Yaskawa INFORM job: A_ROOF_SIDE_0617_2_PAINT_50.JBI

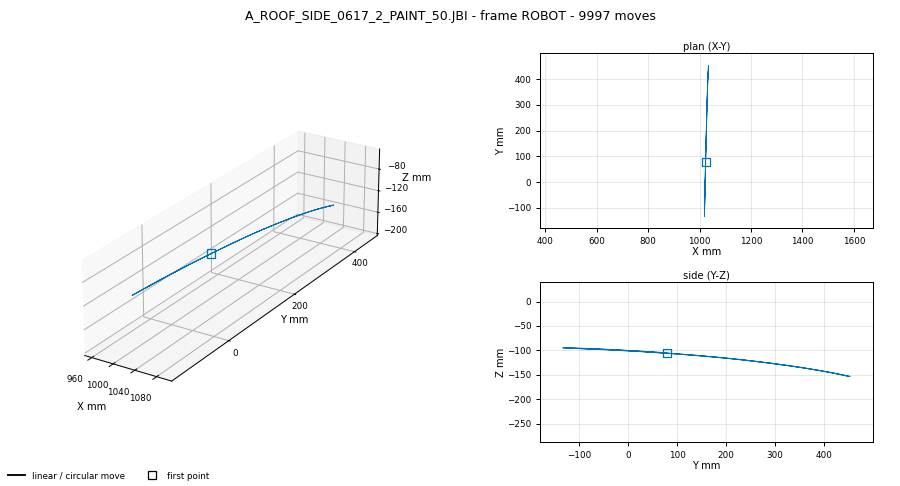
[picture p0: tool path of A_ROOF_SIDE_0617_2_PAINT_50.JBI in frame ROBOT, 9997 of 9997 moves have a stored position in this frame; points joined in program order, loops and branches not executed]
/JOB
//NAME A_ROOF_SIDE_0617_2_PAINT50
//POS
///NPOS 9997,0,0,0,0,0
///TOOL 1
///USER 0
///POSTYPE ROBOT
///RECTAN
///RCONF 1,0,0,0,0,0,0,0,0,0,0,0,0,0,0,0,0,0,0,0,0,0,0,0
C00000=1024.133,78.884,-104.654,167.721,48.501,158.989
C00001=1024.128,78.635,-104.636,167.719,48.505,158.990
C00002=1024.122,78.385,-104.618,167.716,48.509,158.990
C00003=1024.116,78.136,-104.601,167.715,48.513,158.991
C00004=1024.111,77.886,-104.582,167.712,48.517,158.991
C00005=1024.105,77.637,-104.565,167.709,48.522,158.992
C00006=1024.099,77.389,-104.548,167.707,48.526,158.992
C00007=1024.093,77.139,-104.530,167.704,48.530,158.992
C00008=1024.087,76.890,-104.512,167.702,48.535,158.993
C00009=1024.081,76.640,-104.494,167.699,48.539,158.993
C00010=1024.076,76.391,-104.477,167.697,48.543,158.994
C00011=1024.069,76.141,-104.459,167.694,48.547,158.994
C00012=1024.063,75.858,-104.439,167.690,48.552,158.995
C00013=1024.056,75.573,-104.419,167.687,48.558,158.995
C00014=1024.049,75.289,-104.400,167.685,48.562,158.996
C00015=1024.042,75.005,-104.379,167.681,48.567,158.996
C00016=1024.037,74.756,-104.362,167.679,48.572,158.997
C00017=1024.030,74.506,-104.345,167.676,48.576,158.997
C00018=1024.025,74.257,-104.327,167.674,48.580,158.998
C00019=1024.018,74.008,-104.309,167.671,48.585,158.998
C00020=1024.013,73.759,-104.291,167.668,48.589,158.999
C00021=1024.007,73.509,-104.275,167.666,48.593,158.999
C00022=1024.001,73.260,-104.257,167.663,48.597,158.999
C00023=1023.995,73.010,-104.240,167.661,48.602,159.000
C00024=1023.989,72.761,-104.222,167.658,48.606,159.000
C00025=1023.983,72.512,-104.205,167.655,48.610,159.001
C00026=1023.977,72.263,-104.187,167.653,48.614,159.001
C00027=1023.972,72.013,-104.170,167.650,48.619,159.002
C00028=1023.965,71.764,-104.153,167.648,48.623,159.002
C00029=1023.960,71.515,-104.135,167.645,48.627,159.003
C00030=1023.954,71.265,-104.118,167.643,48.632,159.003
C00031=1023.948,71.016,-104.101,167.640,48.636,159.003
C00032=1023.942,70.767,-104.084,167.637,48.640,159.004
C00033=1023.936,70.517,-104.066,167.635,48.644,159.004
C00034=1023.931,70.268,-104.048,167.632,48.649,159.005
C00035=1023.924,70.019,-104.031,167.629,48.653,159.005
C00036=1023.919,69.769,-104.014,167.627,48.657,159.006
C00037=1023.913,69.520,-103.996,167.624,48.661,159.006
C00038=1023.907,69.271,-103.979,167.622,48.666,159.007
C00039=1023.901,69.021,-103.962,167.619,48.670,159.007
C00040=1023.895,68.772,-103.945,167.618,48.674,159.008
C00041=1023.889,68.523,-103.928,167.615,48.678,159.008
C00042=1023.883,68.273,-103.911,167.612,48.682,159.008
C00043=1023.877,68.024,-103.894,167.609,48.687,159.009
C00044=1023.872,67.775,-103.876,167.606,48.691,159.009
C00045=1023.866,67.525,-103.860,167.604,48.696,159.010
C00046=1023.860,67.276,-103.842,167.601,48.700,159.010
C00047=1023.854,67.027,-103.824,167.599,48.704,159.011
C00048=1023.848,66.777,-103.808,167.596,48.709,159.011
C00049=1023.842,66.528,-103.790,167.593,48.713,159.011
C00050=1023.836,66.278,-103.774,167.591,48.717,159.012
C00051=1023.830,66.029,-103.756,167.588,48.721,159.012
C00052=1023.824,65.780,-103.739,167.586,48.726,159.013
C00053=1023.818,65.530,-103.722,167.583,48.730,159.013
C00054=1023.812,65.281,-103.705,167.581,48.734,159.014
C00055=1023.807,65.032,-103.688,167.578,48.738,159.014
C00056=1023.800,64.782,-103.671,167.575,48.743,159.015
C00057=1023.795,64.533,-103.654,167.573,48.748,159.015
C00058=1023.789,64.284,-103.637,167.570,48.752,159.015
C00059=1023.783,64.034,-103.620,167.568,48.756,159.016
C00060=1023.777,63.785,-103.603,167.565,48.760,159.016
C00061=1023.771,63.535,-103.586,167.563,48.765,159.017
C00062=1023.765,63.286,-103.569,167.560,48.769,159.017
C00063=1023.759,63.036,-103.552,167.557,48.773,159.018
C00064=1023.753,62.787,-103.536,167.555,48.778,159.018
C00065=1023.747,62.538,-103.519,167.552,48.782,159.019
C00066=1023.741,62.289,-103.502,167.550,48.786,159.019
C00067=1023.734,62.039,-103.485,167.547,48.791,159.020
C00068=1023.728,61.790,-103.469,167.545,48.796,159.020
C00069=1023.723,61.540,-103.452,167.542,48.799,159.020
C00070=1023.717,61.291,-103.435,167.540,48.804,159.021
C00071=1023.710,61.041,-103.418,167.537,48.809,159.022
C00072=1023.704,60.792,-103.402,167.535,48.813,159.022
C00073=1023.698,60.543,-103.385,167.532,48.817,159.022
C00074=1023.693,60.294,-103.368,167.530,48.822,159.023
C00075=1023.687,60.044,-103.352,167.527,48.826,159.023
C00076=1023.680,59.759,-103.333,167.524,48.831,159.024
C00077=1023.673,59.476,-103.314,167.520,48.836,159.024
C00078=1023.666,59.191,-103.295,167.518,48.841,159.025
C00079=1023.659,58.907,-103.276,167.515,48.846,159.025
C00080=1023.653,58.658,-103.259,167.512,48.850,159.026
C00081=1023.647,58.408,-103.242,167.510,48.855,159.026
C00082=1023.641,58.159,-103.226,167.507,48.860,159.027
C00083=1023.635,57.909,-103.210,167.505,48.864,159.027
C00084=1023.629,57.660,-103.192,167.502,48.868,159.028
C00085=1023.623,57.411,-103.176,167.499,48.872,159.028
C00086=1023.617,57.162,-103.160,167.497,48.877,159.029
C00087=1023.611,56.912,-103.143,167.495,48.881,159.029
C00088=1023.604,56.663,-103.126,167.492,48.885,159.029
C00089=1023.598,56.413,-103.110,167.489,48.890,159.030
C00090=1023.593,56.164,-103.093,167.486,48.895,159.030
C00091=1023.587,55.914,-103.077,167.483,48.899,159.031
C00092=1023.581,55.665,-103.061,167.481,48.903,159.031
C00093=1023.575,55.416,-103.044,167.478,48.907,159.032
C00094=1023.569,55.166,-103.027,167.476,48.912,159.032
C00095=1023.563,54.917,-103.011,167.473,48.917,159.033
C00096=1023.557,54.667,-102.994,167.470,48.921,159.033
C00097=1023.551,54.418,-102.978,167.468,48.925,159.033
C00098=1023.546,54.169,-102.961,167.465,48.929,159.034
C00099=1023.539,53.920,-102.944,167.463,48.934,159.034
C00100=1023.533,53.671,-102.928,167.460,48.938,159.035
C00101=1023.527,53.421,-102.912,167.458,48.942,159.035
C00102=1023.522,53.172,-102.895,167.455,48.946,159.036
C00103=1023.516,52.921,-102.878,167.453,48.951,159.036
C00104=1023.510,52.672,-102.862,167.450,48.955,159.037
C00105=1023.504,52.423,-102.846,167.447,48.959,159.037
C00106=1023.498,52.173,-102.830,167.445,48.964,159.037
C00107=1023.492,51.924,-102.813,167.442,48.968,159.038
C00108=1023.486,51.675,-102.796,167.440,48.973,159.038
C00109=1023.480,51.426,-102.780,167.437,48.977,159.039
C00110=1023.474,51.176,-102.763,167.435,48.981,159.039
C00111=1023.468,50.927,-102.747,167.432,48.985,159.040
C00112=1023.462,50.678,-102.731,167.430,48.990,159.040
C00113=1023.457,50.428,-102.715,167.427,48.994,159.040
C00114=1023.451,50.179,-102.698,167.424,48.998,159.041
C00115=1023.445,49.929,-102.681,167.422,49.002,159.041
C00116=1023.439,49.680,-102.665,167.419,49.007,159.042
C00117=1023.433,49.431,-102.649,167.416,49.011,159.042
C00118=1023.427,49.181,-102.633,167.414,49.016,159.043
C00119=1023.422,48.932,-102.616,167.411,49.019,159.043
C00120=1023.416,48.683,-102.600,167.409,49.024,159.043
C00121=1023.410,48.433,-102.584,167.406,49.028,159.044
C00122=1023.404,48.184,-102.567,167.403,49.032,159.044
C00123=1023.398,47.934,-102.551,167.401,49.037,159.045
C00124=1023.393,47.685,-102.535,167.398,49.041,159.045
C00125=1023.387,47.435,-102.518,167.396,49.045,159.046
C00126=1023.381,47.186,-102.502,167.393,49.049,159.046
C00127=1023.375,46.937,-102.486,167.391,49.054,159.046
C00128=1023.369,46.687,-102.470,167.388,49.058,159.047
C00129=1023.364,46.438,-102.453,167.386,49.062,159.047
C00130=1023.358,46.188,-102.436,167.383,49.066,159.048
C00131=1023.352,45.939,-102.420,167.380,49.070,159.048
C00132=1023.346,45.690,-102.404,167.378,49.075,159.048
C00133=1023.340,45.440,-102.388,167.375,49.079,159.049
C00134=1023.334,45.191,-102.371,167.373,49.084,159.049
C00135=1023.328,44.942,-102.355,167.370,49.087,159.050
C00136=1023.322,44.692,-102.339,167.368,49.091,159.050
C00137=1023.317,44.443,-102.322,167.366,49.096,159.051
C00138=1023.311,44.193,-102.306,167.363,49.100,159.051
C00139=1023.305,43.943,-102.290,167.360,49.104,159.051
C00140=1023.299,43.659,-102.272,167.357,49.109,159.052
C00141=1023.292,43.375,-102.253,167.354,49.113,159.052
C00142=1023.285,43.089,-102.235,167.351,49.118,159.053
C00143=1023.279,42.805,-102.216,167.349,49.123,159.053
C00144=1023.273,42.556,-102.200,167.346,49.128,159.054
C00145=1023.267,42.307,-102.184,167.344,49.132,159.054
C00146=1023.261,42.057,-102.168,167.341,49.136,159.054
C00147=1023.254,41.808,-102.152,167.337,49.140,159.055
C00148=1023.249,41.558,-102.136,167.335,49.145,159.055
C00149=1023.243,41.309,-102.120,167.332,49.149,159.056
C00150=1023.237,41.059,-102.104,167.330,49.154,159.056
C00151=1023.232,40.810,-102.088,167.327,49.158,159.056
C00152=1023.226,40.561,-102.072,167.325,49.162,159.057
C00153=1023.220,40.311,-102.057,167.322,49.166,159.057
C00154=1023.213,40.062,-102.041,167.320,49.171,159.058
C00155=1023.207,39.813,-102.025,167.317,49.175,159.058
C00156=1023.202,39.563,-102.009,167.315,49.180,159.059
C00157=1023.196,39.313,-101.993,167.312,49.183,159.059
C00158=1023.190,39.064,-101.977,167.309,49.188,159.059
C00159=1023.184,38.814,-101.961,167.307,49.192,159.060
C00160=1023.178,38.566,-101.946,167.304,49.197,159.060
C00161=1023.172,38.316,-101.930,167.302,49.201,159.061
C00162=1023.166,38.066,-101.914,167.299,49.205,159.061
C00163=1023.161,37.817,-101.898,167.296,49.209,159.062
C00164=1023.155,37.568,-101.881,167.294,49.213,159.062
C00165=1023.149,37.318,-101.866,167.291,49.218,159.062
C00166=1023.142,37.069,-101.850,167.289,49.222,159.063
C00167=1023.137,36.819,-101.835,167.286,49.227,159.063
C00168=1023.131,36.570,-101.819,167.283,49.231,159.064
C00169=1023.126,36.320,-101.803,167.281,49.235,159.064
C00170=1023.119,36.071,-101.788,167.278,49.239,159.064
C00171=1023.113,35.821,-101.772,167.276,49.244,159.065
C00172=1023.107,35.572,-101.756,167.274,49.249,159.065
C00173=1023.101,35.322,-101.741,167.271,49.253,159.066
C00174=1023.096,35.073,-101.725,167.268,49.257,159.066
C00175=1023.089,34.824,-101.710,167.265,49.261,159.067
C00176=1023.083,34.574,-101.694,167.262,49.266,159.067
C00177=1023.077,34.325,-101.679,167.260,49.270,159.067
C00178=1023.071,34.075,-101.663,167.257,49.275,159.068
C00179=1023.066,33.826,-101.647,167.255,49.279,159.068
C00180=1023.059,33.576,-101.632,167.252,49.283,159.069
C00181=1023.054,33.327,-101.616,167.249,49.287,159.069
C00182=1023.047,33.077,-101.601,167.247,49.292,159.070
C00183=1023.041,32.828,-101.585,167.244,49.296,159.070
C00184=1023.035,32.579,-101.570,167.242,49.301,159.070
C00185=1023.029,32.330,-101.554,167.239,49.305,159.071
C00186=1023.024,32.080,-101.539,167.237,49.309,159.071
C00187=1023.017,31.830,-101.524,167.234,49.313,159.072
C00188=1023.011,31.581,-101.507,167.232,49.318,159.072
C00189=1023.006,31.332,-101.493,167.229,49.322,159.072
C00190=1023.000,31.082,-101.477,167.227,49.327,159.073
C00191=1022.994,30.832,-101.461,167.224,49.331,159.073
C00192=1022.988,30.583,-101.446,167.221,49.336,159.074
C00193=1022.983,30.334,-101.431,167.218,49.340,159.074
C00194=1022.976,30.085,-101.415,167.215,49.344,159.075
C00195=1022.970,29.835,-101.400,167.213,49.348,159.075
C00196=1022.965,29.585,-101.384,167.210,49.352,159.075
C00197=1022.959,29.336,-101.369,167.208,49.357,159.076
C00198=1022.953,29.086,-101.353,167.205,49.361,159.076
C00199=1022.947,28.837,-101.338,167.203,49.366,159.077
C00200=1022.941,28.587,-101.322,167.200,49.370,159.077
C00201=1022.935,28.338,-101.308,167.197,49.374,159.077
C00202=1022.929,28.088,-101.292,167.195,49.378,159.078
C00203=1022.923,27.839,-101.276,167.192,49.382,159.078
C00204=1022.916,27.554,-101.258,167.189,49.387,159.078
C00205=1022.910,27.269,-101.242,167.187,49.393,159.079
C00206=1022.903,26.985,-101.225,167.183,49.398,159.080
C00207=1022.896,26.700,-101.207,167.180,49.403,159.080
C00208=1022.890,26.452,-101.191,167.177,49.407,159.080
C00209=1022.884,26.202,-101.176,167.175,49.411,159.081
C00210=1022.878,25.952,-101.161,167.172,49.415,159.081
C00211=1022.873,25.703,-101.146,167.170,49.420,159.082
C00212=1022.866,25.453,-101.131,167.167,49.424,159.082
C00213=1022.861,25.204,-101.116,167.165,49.429,159.083
C00214=1022.854,24.954,-101.101,167.162,49.433,159.083
C00215=1022.848,24.705,-101.086,167.159,49.437,159.083
C00216=1022.843,24.456,-101.070,167.157,49.441,159.084
C00217=1022.836,24.206,-101.055,167.153,49.446,159.084
C00218=1022.830,23.957,-101.041,167.151,49.450,159.084
C00219=1022.825,23.707,-101.025,167.148,49.455,159.085
C00220=1022.818,23.457,-101.010,167.146,49.459,159.085
C00221=1022.813,23.208,-100.995,167.143,49.464,159.086
C00222=1022.807,22.958,-100.980,167.140,49.468,159.086
C00223=1022.801,22.709,-100.965,167.138,49.472,159.087
C00224=1022.795,22.460,-100.950,167.135,49.476,159.087
C00225=1022.789,22.210,-100.935,167.133,49.481,159.087
C00226=1022.783,21.961,-100.920,167.130,49.485,159.088
C00227=1022.777,21.711,-100.905,167.128,49.490,159.088
C00228=1022.771,21.461,-100.890,167.124,49.494,159.089
C00229=1022.765,21.212,-100.875,167.122,49.498,159.089
C00230=1022.759,20.963,-100.860,167.119,49.503,159.089
C00231=1022.753,20.714,-100.846,167.116,49.507,159.090
C00232=1022.748,20.464,-100.830,167.114,49.511,159.090
C00233=1022.741,20.214,-100.815,167.111,49.515,159.091
C00234=1022.736,19.965,-100.801,167.109,49.519,159.091
C00235=1022.730,19.715,-100.785,167.106,49.524,159.091
C00236=1022.724,19.466,-100.770,167.104,49.528,159.092
C00237=1022.718,19.216,-100.756,167.101,49.533,159.092
C00238=1022.712,18.967,-100.740,167.099,49.537,159.093
C00239=1022.706,18.718,-100.725,167.096,49.541,159.093
C00240=1022.700,18.468,-100.710,167.092,49.546,159.093
C00241=1022.694,18.219,-100.696,167.090,49.550,159.094
C00242=1022.688,17.969,-100.681,167.087,49.554,159.094
C00243=1022.682,17.720,-100.667,167.085,49.559,159.095
C00244=1022.677,17.470,-100.652,167.082,49.563,159.095
C00245=1022.670,17.220,-100.637,167.080,49.567,159.095
C00246=1022.664,16.971,-100.622,167.077,49.572,159.096
C00247=1022.658,16.721,-100.607,167.075,49.576,159.096
C00248=1022.652,16.473,-100.592,167.072,49.581,159.097
C00249=1022.647,16.222,-100.578,167.069,49.585,159.097
C00250=1022.641,15.973,-100.563,167.066,49.590,159.097
C00251=1022.635,15.723,-100.548,167.063,49.594,159.098
C00252=1022.629,15.474,-100.534,167.061,49.598,159.098
C00253=1022.623,15.225,-100.519,167.058,49.602,159.098
C00254=1022.617,14.975,-100.505,167.056,49.606,159.099
C00255=1022.611,14.725,-100.489,167.053,49.611,159.099
C00256=1022.606,14.476,-100.475,167.051,49.615,159.100
C00257=1022.599,14.227,-100.460,167.048,49.619,159.100
C00258=1022.594,13.978,-100.445,167.046,49.624,159.100
C00259=1022.587,13.727,-100.431,167.042,49.628,159.101
C00260=1022.582,13.478,-100.416,167.040,49.633,159.101
C00261=1022.575,13.229,-100.401,167.037,49.637,159.102
C00262=1022.570,12.979,-100.387,167.034,49.642,159.102
C00263=1022.563,12.729,-100.373,167.032,49.646,159.102
C00264=1022.558,12.481,-100.358,167.029,49.650,159.103
C00265=1022.552,12.230,-100.344,167.026,49.655,159.103
C00266=1022.546,11.981,-100.329,167.023,49.659,159.104
C00267=1022.540,11.731,-100.315,167.021,49.663,159.104
C00268=1022.533,11.448,-100.299,167.017,49.668,159.104
C00269=1022.526,11.165,-100.282,167.015,49.674,159.105
C00270=1022.519,10.882,-100.266,167.012,49.679,159.105
C00271=1022.512,10.599,-100.250,167.009,49.684,159.106
C00272=1022.506,10.349,-100.235,167.006,49.688,159.106
C00273=1022.500,10.100,-100.221,167.004,49.693,159.107
C00274=1022.494,9.850,-100.207,167.001,49.697,159.107
C00275=1022.488,9.601,-100.192,166.997,49.702,159.107
C00276=1022.481,9.351,-100.178,166.995,49.706,159.108
C00277=1022.476,9.102,-100.164,166.992,49.710,159.108
C00278=1022.470,8.853,-100.149,166.990,49.714,159.109
C00279=1022.464,8.603,-100.135,166.987,49.719,159.109
C00280=1022.458,8.354,-100.120,166.985,49.723,159.109
C00281=1022.452,8.103,-100.106,166.981,49.728,159.110
C00282=1022.446,7.854,-100.091,166.979,49.732,159.110
C00283=1022.440,7.604,-100.078,166.976,49.737,159.111
C00284=1022.434,7.355,-100.063,166.974,49.741,159.111
C00285=1022.428,7.106,-100.049,166.971,49.745,159.111
C00286=1022.422,6.856,-100.035,166.969,49.750,159.112
C00287=1022.417,6.607,-100.021,166.966,49.754,159.112
C00288=1022.410,6.356,-100.006,166.963,49.759,159.112
C00289=1022.405,6.107,-99.992,166.960,49.763,159.113
C00290=1022.398,5.858,-99.979,166.957,49.767,159.113
C00291=1022.392,5.608,-99.964,166.955,49.771,159.114
C00292=1022.387,5.359,-99.950,166.952,49.775,159.114
C00293=1022.381,5.110,-99.935,166.950,49.780,159.114
C00294=1022.375,4.860,-99.921,166.946,49.785,159.115
C00295=1022.369,4.610,-99.907,166.943,49.789,159.115
C00296=1022.364,4.361,-99.892,166.941,49.793,159.115
C00297=1022.357,4.111,-99.879,166.938,49.797,159.116
C00298=1022.351,3.862,-99.864,166.936,49.802,159.116
C00299=1022.345,3.613,-99.850,166.933,49.806,159.117
C00300=1022.339,3.362,-99.836,166.931,49.810,159.117
C00301=1022.334,3.113,-99.822,166.927,49.815,159.117
C00302=1022.328,2.864,-99.808,166.925,49.819,159.118
C00303=1022.322,2.614,-99.793,166.922,49.823,159.118
C00304=1022.316,2.365,-99.779,166.920,49.828,159.118
C00305=1022.310,2.115,-99.766,166.917,49.832,159.119
C00306=1022.304,1.865,-99.751,166.914,49.836,159.119
C00307=1022.298,1.616,-99.737,166.912,49.841,159.120
C00308=1022.293,1.367,-99.723,166.909,49.845,159.120
C00309=1022.287,1.117,-99.709,166.905,49.849,159.120
C00310=1022.281,0.867,-99.694,166.903,49.854,159.121
C00311=1022.275,0.618,-99.681,166.900,49.858,159.121
C00312=1022.269,0.368,-99.667,166.898,49.862,159.121
C00313=1022.263,0.118,-99.653,166.895,49.866,159.122
C00314=1022.257,-0.131,-99.638,166.893,49.871,159.122
C00315=1022.252,-0.380,-99.624,166.890,49.875,159.122
C00316=1022.246,-0.630,-99.610,166.886,49.879,159.123
C00317=1022.240,-0.880,-99.596,166.884,49.884,159.123
C00318=1022.234,-1.129,-99.582,166.881,49.888,159.123
C00319=1022.228,-1.378,-99.568,166.879,49.892,159.124
C00320=1022.223,-1.628,-99.555,166.876,49.896,159.124
C00321=1022.217,-1.878,-99.541,166.874,49.901,159.125
C00322=1022.211,-2.127,-99.526,166.871,49.905,159.125
C00323=1022.205,-2.377,-99.512,166.868,49.909,159.125
C00324=1022.199,-2.626,-99.499,166.866,49.913,159.125
C00325=1022.194,-2.876,-99.485,166.862,49.917,159.126
C00326=1022.188,-3.125,-99.471,166.860,49.922,159.126
C00327=1022.182,-3.375,-99.456,166.857,49.926,159.127
C00328=1022.176,-3.624,-99.442,166.854,49.930,159.127
C00329=1022.171,-3.874,-99.428,166.851,49.934,159.127
C00330=1022.165,-4.123,-99.415,166.849,49.939,159.128
C00331=1022.159,-4.374,-99.401,166.846,49.943,159.128
C00332=1022.152,-4.654,-99.385,166.843,49.948,159.128
C00333=1022.146,-4.936,-99.370,166.840,49.953,159.129
C00334=1022.139,-5.217,-99.355,166.836,49.958,159.129
C00335=1022.132,-5.499,-99.340,166.834,49.963,159.130
C00336=1022.126,-5.748,-99.326,166.830,49.967,159.130
C00337=1022.120,-5.997,-99.312,166.828,49.972,159.130
C00338=1022.114,-6.247,-99.299,166.825,49.976,159.131
C00339=1022.108,-6.497,-99.285,166.823,49.981,159.131
C00340=1022.102,-6.746,-99.272,166.819,49.985,159.131
C00341=1022.096,-6.996,-99.258,166.817,49.989,159.132
C00342=1022.090,-7.245,-99.244,166.814,49.994,159.132
C00343=1022.085,-7.495,-99.231,166.812,49.998,159.132
C00344=1022.078,-7.745,-99.217,166.809,50.003,159.133
C00345=1022.073,-7.994,-99.203,166.806,50.007,159.133
C00346=1022.066,-8.243,-99.190,166.803,50.011,159.134
C00347=1022.061,-8.493,-99.176,166.801,50.016,159.134
C00348=1022.055,-8.743,-99.163,166.798,50.020,159.134
C00349=1022.049,-8.992,-99.150,166.794,50.024,159.135
C00350=1022.043,-9.242,-99.136,166.792,50.029,159.135
C00351=1022.037,-9.491,-99.123,166.789,50.033,159.135
C00352=1022.031,-9.741,-99.109,166.787,50.037,159.136
C00353=1022.025,-9.991,-99.096,166.784,50.042,159.136
C00354=1022.019,-10.240,-99.082,166.781,50.046,159.136
C00355=1022.013,-10.490,-99.069,166.778,50.050,159.137
C00356=1022.008,-10.740,-99.055,166.776,50.055,159.137
C00357=1022.002,-10.989,-99.042,166.773,50.059,159.137
C00358=1021.996,-11.238,-99.028,166.770,50.063,159.138
C00359=1021.990,-11.488,-99.015,166.767,50.068,159.138
C00360=1021.984,-11.737,-99.001,166.764,50.072,159.138
C00361=1021.979,-11.987,-98.988,166.762,50.076,159.139
C00362=1021.972,-12.236,-98.975,166.759,50.080,159.139
C00363=1021.967,-12.486,-98.961,166.757,50.085,159.140
C00364=1021.961,-12.735,-98.948,166.753,50.090,159.140
C00365=1021.955,-12.985,-98.934,166.750,50.094,159.140
C00366=1021.949,-13.235,-98.922,166.748,50.098,159.140
C00367=1021.943,-13.485,-98.907,166.745,50.102,159.141
C00368=1021.937,-13.734,-98.894,166.743,50.107,159.141
C00369=1021.932,-13.984,-98.880,166.739,50.111,159.141
C00370=1021.926,-14.234,-98.868,166.736,50.115,159.142
C00371=1021.920,-14.483,-98.854,166.734,50.120,159.142
C00372=1021.914,-14.732,-98.841,166.731,50.124,159.143
C00373=1021.908,-14.982,-98.828,166.729,50.128,159.143
C00374=1021.903,-15.232,-98.814,166.725,50.132,159.143
C00375=1021.896,-15.481,-98.801,166.723,50.137,159.144
C00376=1021.891,-15.731,-98.787,166.720,50.141,159.144
C00377=1021.885,-15.981,-98.774,166.717,50.145,159.144
C00378=1021.879,-16.230,-98.761,166.714,50.150,159.145
C00379=1021.873,-16.480,-98.749,166.711,50.154,159.145
C00380=1021.867,-16.729,-98.735,166.709,50.158,159.145
C00381=1021.861,-16.979,-98.722,166.706,50.163,159.146
C00382=1021.855,-17.229,-98.709,166.703,50.168,159.146
C00383=1021.849,-17.478,-98.696,166.700,50.172,159.146
C00384=1021.843,-17.728,-98.683,166.698,50.176,159.147
C00385=1021.837,-17.977,-98.670,166.695,50.180,159.147
C00386=1021.832,-18.226,-98.657,166.691,50.185,159.147
C00387=1021.826,-18.476,-98.644,166.689,50.190,159.148
C00388=1021.820,-18.726,-98.631,166.686,50.194,159.148
C00389=1021.814,-18.975,-98.618,166.683,50.198,159.148
C00390=1021.808,-19.225,-98.605,166.680,50.203,159.149
C00391=1021.803,-19.474,-98.592,166.678,50.207,159.149
C00392=1021.797,-19.724,-98.579,166.675,50.211,159.149
C00393=1021.791,-19.974,-98.566,166.672,50.216,159.150
C00394=1021.785,-20.223,-98.553,166.669,50.220,159.150
C00395=1021.779,-20.473,-98.541,166.666,50.224,159.150
C00396=1021.774,-20.696,-98.529,166.664,50.228,159.151
C00397=1021.768,-20.920,-98.517,166.661,50.232,159.151
C00398=1021.763,-21.143,-98.505,166.658,50.236,159.151
C00399=1021.758,-21.366,-98.495,166.657,50.240,159.152
C00400=1021.753,-21.589,-98.483,166.654,50.244,159.152
C00401=1021.747,-21.813,-98.471,166.651,50.248,159.152
C00402=1021.742,-22.036,-98.459,166.648,50.252,159.152
C00403=1021.737,-22.259,-98.448,166.646,50.256,159.153
C00404=1021.731,-22.509,-98.435,166.643,50.260,159.153
C00405=1021.726,-22.759,-98.422,166.640,50.264,159.153
C00406=1021.719,-23.008,-98.409,166.638,50.269,159.154
C00407=1021.714,-23.258,-98.396,166.634,50.273,159.154
C00408=1021.708,-23.508,-98.384,166.632,50.277,159.154
C00409=1021.702,-23.756,-98.371,166.629,50.281,159.155
C00410=1021.696,-24.006,-98.358,166.627,50.286,159.155
C00411=1021.691,-24.256,-98.345,166.623,50.291,159.155
C00412=1021.685,-24.506,-98.332,166.620,50.295,159.156
C00413=1021.679,-24.756,-98.319,166.618,50.299,159.156
C00414=1021.673,-25.006,-98.307,166.616,50.303,159.156
C00415=1021.667,-25.254,-98.294,166.612,50.308,159.157
C00416=1021.661,-25.504,-98.281,166.609,50.312,159.157
C00417=1021.655,-25.754,-98.269,166.607,50.316,159.157
C00418=1021.650,-26.003,-98.255,166.604,50.320,159.157
C00419=1021.644,-26.253,-98.242,166.600,50.325,159.158
C00420=1021.639,-26.502,-98.230,166.598,50.329,159.158
C00421=1021.633,-26.752,-98.217,166.595,50.333,159.158
C00422=1021.627,-27.002,-98.204,166.593,50.337,159.159
C00423=1021.621,-27.252,-98.192,166.590,50.342,159.159
C00424=1021.615,-27.501,-98.179,166.586,50.346,159.159
C00425=1021.610,-27.751,-98.167,166.584,50.351,159.160
C00426=1021.604,-28.000,-98.154,166.581,50.355,159.160
C00427=1021.597,-28.250,-98.141,166.578,50.359,159.160
C00428=1021.591,-28.500,-98.129,166.575,50.364,159.161
C00429=1021.586,-28.749,-98.116,166.573,50.368,159.161
C00430=1021.580,-28.999,-98.104,166.569,50.373,159.161
C00431=1021.574,-29.249,-98.091,166.567,50.377,159.162
C00432=1021.568,-29.498,-98.079,166.564,50.381,159.162
C00433=1021.562,-29.748,-98.067,166.560,50.386,159.162
C00434=1021.557,-29.997,-98.055,166.558,50.391,159.163
C00435=1021.551,-30.247,-98.042,166.555,50.395,159.163
C00436=1021.543,-30.579,-98.025,166.551,50.401,159.163
C00437=1021.535,-30.911,-98.009,166.547,50.406,159.164
C00438=1021.527,-31.244,-97.992,166.543,50.412,159.164
C00439=1021.519,-31.576,-97.976,166.540,50.418,159.165
C00440=1021.514,-31.825,-97.964,166.537,50.423,159.165
C00441=1021.508,-32.075,-97.951,166.534,50.427,159.165
C00442=1021.502,-32.325,-97.939,166.531,50.431,159.166
C00443=1021.496,-32.574,-97.927,166.528,50.436,159.166
C00444=1021.490,-32.824,-97.914,166.525,50.440,159.166
C00445=1021.484,-33.074,-97.902,166.523,50.444,159.166
C00446=1021.478,-33.324,-97.889,166.520,50.448,159.167
C00447=1021.473,-33.573,-97.877,166.517,50.453,159.167
C00448=1021.467,-33.823,-97.864,166.514,50.458,159.167
C00449=1021.461,-34.072,-97.852,166.511,50.462,159.168
C00450=1021.455,-34.321,-97.840,166.508,50.466,159.168
C00451=1021.449,-34.571,-97.828,166.505,50.470,159.168
C00452=1021.444,-34.821,-97.816,166.503,50.475,159.169
C00453=1021.438,-35.070,-97.803,166.499,50.479,159.169
C00454=1021.432,-35.320,-97.790,166.496,50.483,159.169
C00455=1021.427,-35.569,-97.778,166.494,50.488,159.170
C00456=1021.420,-35.819,-97.766,166.491,50.492,159.170
C00457=1021.415,-36.070,-97.754,166.488,50.497,159.170
C00458=1021.409,-36.319,-97.742,166.485,50.501,159.170
C00459=1021.404,-36.569,-97.730,166.483,50.505,159.171
C00460=1021.397,-36.847,-97.716,166.479,50.509,159.171
C00461=1021.391,-37.126,-97.702,166.476,50.515,159.171
C00462=1021.384,-37.404,-97.689,166.472,50.520,159.172
C00463=1021.378,-37.682,-97.675,166.470,50.524,159.172
C00464=1021.372,-37.933,-97.663,166.466,50.528,159.172
C00465=1021.366,-38.183,-97.651,166.464,50.533,159.173
C00466=1021.361,-38.432,-97.639,166.461,50.537,159.173
C00467=1021.355,-38.682,-97.626,166.457,50.542,159.173
C00468=1021.350,-38.931,-97.614,166.455,50.546,159.173
C00469=1021.343,-39.181,-97.603,166.452,50.550,159.174
C00470=1021.338,-39.430,-97.591,166.448,50.554,159.174
C00471=1021.332,-39.680,-97.578,166.446,50.559,159.174
C00472=1021.326,-39.930,-97.567,166.443,50.563,159.175
C00473=1021.321,-40.180,-97.555,166.440,50.568,159.175
C00474=1021.314,-40.429,-97.543,166.437,50.572,159.175
C00475=1021.309,-40.679,-97.531,166.435,50.577,159.176
C00476=1021.303,-40.929,-97.519,166.431,50.581,159.176
C00477=1021.297,-41.178,-97.507,166.429,50.585,159.176
C00478=1021.291,-41.428,-97.495,166.426,50.590,159.177
C00479=1021.285,-41.677,-97.484,166.423,50.594,159.177
C00480=1021.279,-41.927,-97.471,166.420,50.598,159.177
C00481=1021.274,-42.176,-97.460,166.416,50.603,159.177
C00482=1021.268,-42.426,-97.448,166.414,50.608,159.178
C00483=1021.263,-42.676,-97.436,166.411,50.612,159.178
C00484=1021.256,-42.926,-97.424,166.408,50.616,159.178
C00485=1021.251,-43.175,-97.412,166.405,50.620,159.179
C00486=1021.244,-43.425,-97.401,166.402,50.625,159.179
C00487=1021.239,-43.674,-97.389,166.399,50.630,159.179
C00488=1021.233,-43.924,-97.377,166.397,50.634,159.179
C00489=1021.228,-44.174,-97.365,166.394,50.638,159.180
C00490=1021.221,-44.424,-97.354,166.390,50.642,159.180
C00491=1021.216,-44.673,-97.342,166.388,50.646,159.180
C00492=1021.210,-44.924,-97.330,166.385,50.651,159.181
C00493=1021.204,-45.172,-97.318,166.382,50.656,159.181
C00494=1021.199,-45.422,-97.307,166.379,50.660,159.181
C00495=1021.193,-45.672,-97.295,166.375,50.664,159.181
C00496=1021.188,-45.922,-97.283,166.373,50.668,159.182
C00497=1021.181,-46.171,-97.271,166.370,50.673,159.182
C00498=1021.176,-46.421,-97.260,166.367,50.678,159.182
C00499=1021.169,-46.671,-97.248,166.364,50.682,159.183
C00500=1021.164,-46.920,-97.236,166.362,50.686,159.183
C00501=1021.159,-47.169,-97.224,166.358,50.690,159.183
C00502=1021.153,-47.420,-97.213,166.355,50.694,159.183
C00503=1021.148,-47.669,-97.202,166.353,50.699,159.184
C00504=1021.141,-47.919,-97.190,166.349,50.703,159.184
C00505=1021.136,-48.169,-97.178,166.347,50.708,159.184
C00506=1021.130,-48.418,-97.167,166.344,50.712,159.185
C00507=1021.124,-48.668,-97.155,166.340,50.716,159.185
C00508=1021.118,-48.917,-97.143,166.338,50.721,159.185
C00509=1021.113,-49.167,-97.132,166.335,50.725,159.185
C00510=1021.107,-49.417,-97.120,166.331,50.729,159.186
C00511=1021.102,-49.666,-97.108,166.329,50.733,159.186
C00512=1021.096,-49.916,-97.097,166.326,50.737,159.186
C00513=1021.090,-50.166,-97.086,166.322,50.742,159.186
C00514=1021.085,-50.415,-97.073,166.320,50.746,159.187
C00515=1021.079,-50.665,-97.062,166.317,50.750,159.187
C00516=1021.074,-50.915,-97.051,166.314,50.755,159.187
C00517=1021.068,-51.164,-97.039,166.311,50.759,159.188
C00518=1021.062,-51.414,-97.028,166.309,50.764,159.188
C00519=1021.056,-51.664,-97.017,166.305,50.769,159.188
C00520=1021.050,-51.913,-97.006,166.303,50.773,159.188
C00521=1021.044,-52.163,-96.995,166.299,50.777,159.189
C00522=1021.038,-52.413,-96.983,166.297,50.782,159.189
C00523=1021.033,-52.663,-96.972,166.293,50.787,159.189
C00524=1021.026,-52.942,-96.960,166.290,50.792,159.190
C00525=1021.019,-53.221,-96.948,166.287,50.797,159.190
C00526=1021.013,-53.500,-96.935,166.283,50.801,159.190
C00527=1021.006,-53.778,-96.923,166.280,50.807,159.191
C00528=1021.000,-54.029,-96.911,166.277,50.811,159.191
C00529=1020.995,-54.278,-96.900,166.274,50.816,159.191
C00530=1020.989,-54.528,-96.889,166.271,50.820,159.191
C00531=1020.983,-54.777,-96.878,166.267,50.825,159.192
C00532=1020.977,-55.027,-96.867,166.265,50.829,159.192
C00533=1020.971,-55.277,-96.856,166.263,50.834,159.192
C00534=1020.965,-55.526,-96.845,166.259,50.838,159.193
C00535=1020.960,-55.776,-96.834,166.256,50.842,159.193
C00536=1020.954,-56.026,-96.822,166.253,50.847,159.193
C00537=1020.948,-56.276,-96.812,166.250,50.851,159.194
C00538=1020.943,-56.525,-96.801,166.247,50.856,159.194
C00539=1020.937,-56.775,-96.790,166.244,50.860,159.194
C00540=1020.931,-57.025,-96.779,166.241,50.865,159.194
C00541=1020.925,-57.275,-96.768,166.238,50.869,159.195
C00542=1020.919,-57.524,-96.757,166.236,50.873,159.195
C00543=1020.913,-57.773,-96.746,166.232,50.878,159.195
C00544=1020.908,-58.023,-96.735,166.230,50.883,159.196
C00545=1020.902,-58.273,-96.723,166.226,50.887,159.196
///RCONF 1,0,0,1,0,0,0,0,0,0,0,0,0,0,0,0,0,0,0,0,0,0,0,0
C00546=1020.896,-58.523,-96.712,166.223,50.891,159.196
C00547=1020.890,-58.772,-96.702,166.220,50.896,159.196
C00548=1020.885,-59.022,-96.691,166.217,50.900,159.196
C00549=1020.879,-59.271,-96.680,166.215,50.905,159.197
C00550=1020.873,-59.521,-96.669,166.211,50.909,159.197
C00551=1020.867,-59.771,-96.658,166.209,50.914,159.197
C00552=1020.862,-60.021,-96.646,166.205,50.918,159.198
C00553=1020.856,-60.271,-96.636,166.202,50.922,159.198
C00554=1020.851,-60.521,-96.625,166.199,50.927,159.198
C00555=1020.845,-60.770,-96.614,166.196,50.931,159.198
C00556=1020.839,-61.020,-96.603,166.194,50.936,159.199
C00557=1020.834,-61.269,-96.592,166.190,50.940,159.199
C00558=1020.828,-61.518,-96.582,166.188,50.944,159.199
C00559=1020.821,-61.769,-96.570,166.184,50.949,159.199
C00560=1020.816,-62.019,-96.560,166.181,50.953,159.200
C00561=1020.810,-62.268,-96.549,166.179,50.957,159.200
C00562=1020.805,-62.518,-96.538,166.175,50.962,159.200
C00563=1020.800,-62.768,-96.527,166.173,50.966,159.201
C00564=1020.794,-63.017,-96.516,166.169,50.971,159.201
C00565=1020.788,-63.267,-96.505,166.167,50.975,159.201
C00566=1020.783,-63.517,-96.495,166.164,50.979,159.201
C00567=1020.777,-63.766,-96.484,166.160,50.984,159.201
C00568=1020.771,-64.016,-96.473,166.158,50.988,159.202
C00569=1020.765,-64.265,-96.462,166.154,50.992,159.202
C00570=1020.760,-64.515,-96.452,166.151,50.996,159.202
C00571=1020.754,-64.765,-96.441,166.149,51.001,159.203
C00572=1020.749,-65.015,-96.430,166.145,51.006,159.203
C00573=1020.743,-65.264,-96.419,166.143,51.010,159.203
C00574=1020.738,-65.514,-96.409,166.139,51.014,159.203
C00575=1020.732,-65.764,-96.398,166.137,51.019,159.204
C00576=1020.727,-66.013,-96.387,166.134,51.023,159.204
C00577=1020.721,-66.263,-96.377,166.130,51.027,159.204
C00578=1020.715,-66.513,-96.366,166.128,51.031,159.204
C00579=1020.710,-66.762,-96.355,166.124,51.036,159.204
C00580=1020.704,-67.012,-96.344,166.121,51.040,159.205
C00581=1020.698,-67.262,-96.334,166.119,51.044,159.205
C00582=1020.693,-67.511,-96.323,166.115,51.049,159.205
C00583=1020.687,-67.761,-96.312,166.113,51.053,159.205
C00584=1020.682,-68.011,-96.302,166.109,51.057,159.206
C00585=1020.677,-68.261,-96.291,166.106,51.061,159.206
C00586=1020.671,-68.511,-96.281,166.104,51.066,159.206
C00587=1020.665,-68.760,-96.270,166.100,51.070,159.206
C00588=1020.659,-69.041,-96.257,166.097,51.075,159.207
C00589=1020.653,-69.321,-96.246,166.094,51.080,159.207
C00590=1020.647,-69.601,-96.234,166.091,51.085,159.207
C00591=1020.641,-69.881,-96.222,166.087,51.089,159.207
C00592=1020.635,-70.131,-96.212,166.084,51.094,159.208
C00593=1020.629,-70.380,-96.201,166.081,51.098,159.208
C00594=1020.624,-70.630,-96.190,166.078,51.102,159.208
C00595=1020.618,-70.880,-96.180,166.075,51.107,159.208
C00596=1020.613,-71.130,-96.169,166.072,51.111,159.209
C00597=1020.607,-71.380,-96.159,166.070,51.115,159.209
C00598=1020.602,-71.628,-96.148,166.066,51.119,159.209
C00599=1020.596,-71.878,-96.138,166.063,51.124,159.209
C00600=1020.591,-72.128,-96.127,166.061,51.128,159.210
C00601=1020.585,-72.378,-96.117,166.057,51.132,159.210
C00602=1020.580,-72.628,-96.106,166.054,51.136,159.210
C00603=1020.574,-72.878,-96.096,166.050,51.140,159.210
C00604=1020.568,-73.127,-96.085,166.048,51.144,159.210
C00605=1020.564,-73.377,-96.075,166.045,51.148,159.211
C00606=1020.558,-73.626,-96.064,166.042,51.153,159.211
C00607=1020.553,-73.876,-96.053,166.039,51.157,159.211
C00608=1020.548,-74.127,-96.043,166.036,51.161,159.211
C00609=1020.542,-74.376,-96.032,166.033,51.166,159.211
C00610=1020.536,-74.626,-96.023,166.030,51.170,159.212
C00611=1020.531,-74.875,-96.013,166.027,51.174,159.212
C00612=1020.525,-75.125,-96.002,166.024,51.179,159.212
C00613=1020.520,-75.375,-95.992,166.021,51.183,159.212
C00614=1020.514,-75.625,-95.982,166.018,51.187,159.213
C00615=1020.508,-75.874,-95.972,166.015,51.192,159.213
C00616=1020.502,-76.124,-95.961,166.012,51.197,159.213
C00617=1020.498,-76.374,-95.952,166.009,51.201,159.213
C00618=1020.492,-76.624,-95.941,166.005,51.205,159.214
C00619=1020.486,-76.873,-95.931,166.003,51.210,159.214
C00620=1020.480,-77.123,-95.921,166.000,51.214,159.214
C00621=1020.475,-77.372,-95.911,165.997,51.218,159.214
C00622=1020.470,-77.623,-95.901,165.994,51.223,159.215
C00623=1020.463,-77.872,-95.891,165.990,51.227,159.215
C00624=1020.458,-78.122,-95.881,165.988,51.231,159.215
C00625=1020.453,-78.372,-95.870,165.984,51.236,159.215
C00626=1020.448,-78.621,-95.861,165.982,51.240,159.215
C00627=1020.442,-78.871,-95.851,165.979,51.244,159.216
C00628=1020.436,-79.121,-95.840,165.975,51.249,159.216
C00629=1020.431,-79.370,-95.830,165.973,51.253,159.216
C00630=1020.426,-79.620,-95.820,165.969,51.257,159.216
C00631=1020.419,-79.870,-95.811,165.966,51.261,159.216
C00632=1020.414,-80.120,-95.801,165.963,51.266,159.217
C00633=1020.409,-80.369,-95.791,165.960,51.270,159.217
C00634=1020.403,-80.619,-95.781,165.957,51.275,159.217
C00635=1020.398,-80.869,-95.771,165.954,51.280,159.218
C00636=1020.391,-81.119,-95.761,165.951,51.284,159.218
C00637=1020.387,-81.369,-95.752,165.948,51.288,159.218
C00638=1020.380,-81.618,-95.742,165.945,51.293,159.218
C00639=1020.375,-81.868,-95.732,165.942,51.298,159.219
C00640=1020.369,-82.118,-95.723,165.939,51.302,159.219
C00641=1020.363,-82.367,-95.713,165.936,51.306,159.219
C00642=1020.358,-82.617,-95.703,165.932,51.311,159.219
C00643=1020.352,-82.867,-95.694,165.930,51.315,159.219
C00644=1020.347,-83.117,-95.684,165.926,51.320,159.220
C00645=1020.341,-83.366,-95.674,165.924,51.324,159.220
C00646=1020.336,-83.616,-95.664,165.920,51.329,159.220
C00647=1020.330,-83.866,-95.655,165.918,51.333,159.220
C00648=1020.324,-84.116,-95.645,165.914,51.338,159.221
C00649=1020.319,-84.365,-95.635,165.912,51.342,159.221
C00650=1020.313,-84.615,-95.625,165.908,51.346,159.221
C00651=1020.308,-84.865,-95.617,165.905,51.351,159.221
C00652=1020.301,-85.147,-95.605,165.902,51.356,159.222
C00653=1020.295,-85.429,-95.594,165.899,51.361,159.222
C00654=1020.289,-85.711,-95.584,165.895,51.366,159.222
C00655=1020.283,-85.994,-95.573,165.892,51.371,159.222
C00656=1020.277,-86.243,-95.563,165.888,51.375,159.223
C00657=1020.272,-86.493,-95.553,165.886,51.380,159.223
C00658=1020.266,-86.743,-95.545,165.882,51.384,159.223
C00659=1020.261,-86.993,-95.534,165.880,51.388,159.223
C00660=1020.255,-87.243,-95.525,165.876,51.393,159.223
C00661=1020.250,-87.492,-95.515,165.873,51.397,159.224
C00662=1020.244,-87.742,-95.506,165.870,51.402,159.224
C00663=1020.238,-87.991,-95.496,165.867,51.407,159.224
C00664=1020.233,-88.242,-95.487,165.865,51.411,159.225
C00665=1020.227,-88.491,-95.478,165.861,51.415,159.225
C00666=1020.222,-88.741,-95.468,165.859,51.419,159.225
C00667=1020.216,-88.990,-95.458,165.855,51.424,159.225
C00668=1020.211,-89.241,-95.449,165.852,51.428,159.225
C00669=1020.206,-89.490,-95.440,165.849,51.433,159.225
C00670=1020.200,-89.740,-95.430,165.846,51.437,159.226
C00671=1020.195,-89.989,-95.420,165.843,51.441,159.226
C00672=1020.189,-90.239,-95.411,165.840,51.446,159.226
C00673=1020.184,-90.489,-95.402,165.836,51.450,159.226
C00674=1020.178,-90.739,-95.392,165.834,51.454,159.227
C00675=1020.173,-90.989,-95.383,165.831,51.459,159.227
C00676=1020.167,-91.238,-95.373,165.828,51.463,159.227
C00677=1020.162,-91.488,-95.364,165.825,51.467,159.227
C00678=1020.156,-91.738,-95.355,165.821,51.472,159.227
C00679=1020.151,-91.987,-95.346,165.819,51.476,159.228
C00680=1020.145,-92.237,-95.335,165.815,51.481,159.228
C00681=1020.140,-92.487,-95.327,165.813,51.485,159.228
C00682=1020.135,-92.737,-95.317,165.810,51.489,159.228
C00683=1020.129,-92.986,-95.308,165.806,51.494,159.228
C00684=1020.125,-93.236,-95.299,165.804,51.498,159.229
C00685=1020.118,-93.486,-95.289,165.800,51.502,159.229
C00686=1020.113,-93.736,-95.280,165.798,51.507,159.229
C00687=1020.108,-93.986,-95.270,165.794,51.511,159.229
C00688=1020.102,-94.235,-95.261,165.791,51.515,159.229
C00689=1020.098,-94.485,-95.252,165.789,51.520,159.230
C00690=1020.091,-94.735,-95.242,165.785,51.523,159.230
C00691=1020.087,-94.985,-95.233,165.782,51.528,159.230
C00692=1020.081,-95.235,-95.224,165.778,51.532,159.230
C00693=1020.076,-95.484,-95.215,165.776,51.536,159.230
C00694=1020.071,-95.734,-95.206,165.773,51.541,159.231
C00695=1020.065,-95.984,-95.196,165.770,51.545,159.231
C00696=1020.060,-96.234,-95.187,165.767,51.549,159.231
C00697=1020.054,-96.483,-95.178,165.763,51.554,159.231
C00698=1020.049,-96.733,-95.169,165.761,51.558,159.231
C00699=1020.044,-96.983,-95.159,165.758,51.562,159.232
C00700=1020.038,-97.232,-95.151,165.755,51.567,159.232
C00701=1020.033,-97.482,-95.140,165.752,51.570,159.232
C00702=1020.028,-97.732,-95.132,165.748,51.575,159.232
C00703=1020.022,-97.983,-95.123,165.745,51.579,159.232
C00704=1020.017,-98.232,-95.113,165.742,51.584,159.232
C00705=1020.012,-98.482,-95.105,165.739,51.588,159.233
C00706=1020.006,-98.732,-95.096,165.736,51.593,159.233
C00707=1020.000,-98.981,-95.087,165.733,51.597,159.233
C00708=1019.995,-99.231,-95.078,165.730,51.602,159.233
C00709=1019.990,-99.481,-95.070,165.727,51.606,159.234
C00710=1019.984,-99.730,-95.060,165.725,51.610,159.234
C00711=1019.979,-99.980,-95.051,165.721,51.615,159.234
C00712=1019.974,-100.230,-95.043,165.719,51.619,159.234
C00713=1019.968,-100.481,-95.034,165.715,51.624,159.234
C00714=1019.962,-100.730,-95.025,165.712,51.628,159.235
C00715=1019.957,-100.979,-95.016,165.709,51.632,159.235
C00716=1019.951,-101.264,-95.006,165.705,51.638,159.235
C00717=1019.945,-101.548,-94.997,165.702,51.642,159.235
C00718=1019.939,-101.832,-94.986,165.699,51.648,159.236
C00719=1019.933,-102.117,-94.976,165.695,51.652,159.236
C00720=1019.927,-102.366,-94.967,165.691,51.657,159.236
C00721=1019.922,-102.616,-94.959,165.689,51.661,159.236
C00722=1019.916,-102.866,-94.950,165.685,51.665,159.236
C00723=1019.911,-103.116,-94.941,165.683,51.670,159.236
C00724=1019.905,-103.365,-94.932,165.680,51.674,159.237
C00725=1019.901,-103.615,-94.923,165.676,51.678,159.237
C00726=1019.896,-103.865,-94.914,165.674,51.683,159.237
C00727=1019.890,-104.115,-94.906,165.670,51.687,159.237
C00728=1019.884,-104.365,-94.897,165.668,51.691,159.238
C00729=1019.879,-104.614,-94.888,165.664,51.696,159.238
C00730=1019.874,-104.864,-94.879,165.661,51.700,159.238
C00731=1019.868,-105.114,-94.871,165.658,51.705,159.238
C00732=1019.863,-105.363,-94.863,165.655,51.709,159.238
C00733=1019.857,-105.614,-94.854,165.653,51.713,159.239
C00734=1019.852,-105.864,-94.845,165.649,51.718,159.239
C00735=1019.847,-106.113,-94.837,165.647,51.722,159.239
C00736=1019.842,-106.363,-94.828,165.643,51.727,159.239
C00737=1019.837,-106.613,-94.819,165.640,51.731,159.239
C00738=1019.832,-106.863,-94.811,165.637,51.735,159.239
C00739=1019.826,-107.112,-94.802,165.634,51.740,159.240
C00740=1019.820,-107.363,-94.793,165.631,51.744,159.240
C00741=1019.815,-107.613,-94.785,165.628,51.748,159.240
C00742=1019.810,-107.862,-94.776,165.625,51.753,159.240
C00743=1019.805,-108.112,-94.768,165.622,51.757,159.240
C00744=1019.799,-108.362,-94.759,165.619,51.762,159.241
C00745=1019.794,-108.611,-94.751,165.616,51.766,159.241
C00746=1019.788,-108.861,-94.743,165.613,51.770,159.241
C00747=1019.783,-109.111,-94.734,165.609,51.775,159.241
C00748=1019.778,-109.360,-94.726,165.607,51.779,159.241
C00749=1019.772,-109.610,-94.718,165.603,51.784,159.242
C00750=1019.766,-109.860,-94.709,165.601,51.788,159.242
C00751=1019.761,-110.110,-94.700,165.597,51.793,159.242
C00752=1019.756,-110.360,-94.692,165.594,51.797,159.242
C00753=1019.751,-110.610,-94.684,165.591,51.801,159.242
C00754=1019.746,-110.860,-94.675,165.588,51.806,159.243
C00755=1019.740,-111.110,-94.667,165.586,51.810,159.243
C00756=1019.735,-111.359,-94.658,165.582,51.814,159.243
C00757=1019.729,-111.609,-94.651,165.580,51.819,159.243
C00758=1019.724,-111.858,-94.642,165.576,51.823,159.243
C00759=1019.719,-112.108,-94.634,165.573,51.827,159.244
C00760=1019.714,-112.358,-94.626,165.570,51.832,159.244
C00761=1019.708,-112.608,-94.617,165.567,51.836,159.244
C00762=1019.703,-112.858,-94.609,165.564,51.841,159.244
C00763=1019.698,-113.108,-94.600,165.561,51.845,159.244
C00764=1019.693,-113.357,-94.592,165.558,51.849,159.245
C00765=1019.688,-113.608,-94.584,165.555,51.854,159.245
C00766=1019.682,-113.857,-94.576,165.552,51.858,159.245
C00767=1019.676,-114.107,-94.568,165.549,51.863,159.245
C00768=1019.671,-114.356,-94.559,165.546,51.867,159.245
C00769=1019.666,-114.607,-94.552,165.542,51.872,159.245
C00770=1019.661,-114.857,-94.543,165.540,51.876,159.246
C00771=1019.656,-115.106,-94.535,165.536,51.880,159.246
C00772=1019.650,-115.356,-94.527,165.534,51.885,159.246
C00773=1019.645,-115.606,-94.519,165.531,51.889,159.246
C00774=1019.640,-115.855,-94.511,165.528,51.893,159.246
C00775=1019.635,-116.105,-94.503,165.525,51.898,159.247
C00776=1019.630,-116.355,-94.495,165.521,51.902,159.247
C00777=1019.624,-116.604,-94.487,165.519,51.907,159.247
C00778=1019.619,-116.855,-94.479,165.515,51.911,159.247
C00779=1019.614,-117.104,-94.470,165.513,51.915,159.247
C00780=1019.608,-117.389,-94.461,165.509,51.920,159.248
C00781=1019.602,-117.672,-94.453,165.506,51.925,159.248
C00782=1019.595,-117.957,-94.443,165.502,51.930,159.248
C00783=1019.590,-118.242,-94.434,165.499,51.935,159.248
C00784=1019.584,-118.491,-94.426,165.495,51.940,159.248
C00785=1019.579,-118.741,-94.418,165.493,51.944,159.249
C00786=1019.574,-118.990,-94.410,165.489,51.949,159.249
C00787=1019.569,-119.241,-94.402,165.487,51.953,159.249
C00788=1019.563,-119.490,-94.394,165.483,51.957,159.249
C00789=1019.558,-119.740,-94.387,165.481,51.962,159.249
C00790=1019.553,-119.990,-94.378,165.478,51.966,159.250
C00791=1019.547,-120.240,-94.371,165.474,51.971,159.250
C00792=1019.542,-120.490,-94.363,165.472,51.975,159.250
C00793=1019.538,-120.739,-94.355,165.468,51.979,159.250
C00794=1019.532,-120.989,-94.347,165.466,51.984,159.250
C00795=1019.527,-121.239,-94.339,165.462,51.988,159.250
C00796=1019.521,-121.489,-94.331,165.459,51.993,159.251
C00797=1019.516,-121.739,-94.324,165.457,51.996,159.251
C00798=1019.511,-121.988,-94.316,165.453,52.001,159.251
C00799=1019.506,-122.238,-94.308,165.450,52.005,159.251
C00800=1019.500,-122.488,-94.301,165.447,52.010,159.251
C00801=1019.495,-122.738,-94.292,165.444,52.014,159.251
C00802=1019.490,-122.988,-94.284,165.441,52.018,159.252
C00803=1019.485,-123.237,-94.277,165.438,52.023,159.252
C00804=1019.480,-123.487,-94.269,165.436,52.027,159.252
C00805=1019.475,-123.738,-94.261,165.432,52.032,159.252
C00806=1019.469,-123.987,-94.254,165.429,52.036,159.252
C00807=1019.464,-124.237,-94.246,165.426,52.040,159.253
C00808=1019.459,-124.487,-94.238,165.423,52.045,159.253
C00809=1019.453,-124.736,-94.230,165.421,52.049,159.253
C00810=1019.448,-124.987,-94.223,165.417,52.054,159.253
C00811=1019.443,-125.236,-94.216,165.414,52.058,159.253
C00812=1019.438,-125.486,-94.208,165.411,52.062,159.253
C00813=1019.432,-125.736,-94.200,165.408,52.067,159.254
C00814=1019.428,-125.986,-94.193,165.405,52.071,159.254
C00815=1019.422,-126.236,-94.186,165.402,52.076,159.254
C00816=1019.417,-126.486,-94.178,165.400,52.080,159.254
C00817=1019.411,-126.735,-94.170,165.396,52.084,159.254
C00818=1019.407,-126.985,-94.163,165.393,52.089,159.255
C00819=1019.401,-127.235,-94.155,165.390,52.093,159.255
C00820=1019.397,-127.485,-94.148,165.387,52.098,159.255
C00821=1019.391,-127.734,-94.140,165.384,52.102,159.255
C00822=1019.387,-127.984,-94.133,165.381,52.106,159.255
C00823=1019.382,-128.234,-94.125,165.378,52.110,159.255
C00824=1019.377,-128.483,-94.117,165.375,52.114,159.255
C00825=1019.372,-128.733,-94.108,165.372,52.117,159.255
C00826=1019.369,-128.982,-94.098,165.370,52.120,159.255
C00827=1019.367,-129.232,-94.088,165.367,52.121,159.255
C00828=1019.363,-129.482,-94.077,165.364,52.123,159.255
C00829=1019.361,-129.732,-94.066,165.361,52.124,159.255
C00830=1019.359,-129.981,-94.054,165.359,52.125,159.254
C00831=1019.358,-130.231,-94.041,165.357,52.125,159.254
C00832=1019.357,-130.481,-94.028,165.355,52.124,159.253
C00833=1019.357,-130.730,-94.015,165.352,52.123,159.253
C00834=1019.356,-130.979,-94.001,165.350,52.122,159.252
C00835=1019.357,-131.229,-93.986,165.348,52.120,159.251
C00836=1019.358,-131.479,-93.970,165.346,52.117,159.250
C00837=1019.359,-131.729,-93.954,165.344,52.113,159.249
C00838=1019.360,-131.979,-93.937,165.342,52.110,159.249
C00839=1019.363,-132.228,-93.920,165.340,52.106,159.247
C00840=1019.366,-132.478,-93.902,165.338,52.101,159.246
C00841=1019.369,-132.729,-93.884,165.337,52.096,159.245
C00842=1019.372,-132.977,-93.866,165.335,52.090,159.244
C00843=1019.376,-133.228,-93.846,165.334,52.084,159.242
C00844=1019.105,-133.253,-94.214,165.290,52.401,159.288
C00845=1019.100,-133.004,-94.234,165.292,52.407,159.290
C00846=1019.097,-132.755,-94.252,165.294,52.413,159.291
C00847=1019.094,-132.505,-94.270,165.296,52.418,159.292
C00848=1019.091,-132.254,-94.288,165.298,52.423,159.294
C00849=1019.089,-132.005,-94.305,165.299,52.427,159.294
C00850=1019.087,-131.756,-94.322,165.301,52.430,159.296
C00851=1019.085,-131.506,-94.339,165.303,52.433,159.296
C00852=1019.085,-131.256,-94.354,165.305,52.436,159.297
C00853=1019.085,-131.006,-94.368,165.308,52.438,159.298
C00854=1019.084,-130.757,-94.383,165.310,52.440,159.299
C00855=1019.085,-130.507,-94.396,165.312,52.441,159.299
C00856=1019.086,-130.257,-94.409,165.314,52.441,159.300
C00857=1019.087,-130.007,-94.423,165.317,52.441,159.300
C00858=1019.089,-129.757,-94.434,165.319,52.440,159.301
C00859=1019.091,-129.508,-94.445,165.321,52.439,159.301
C00860=1019.094,-129.258,-94.456,165.324,52.438,159.301
C00861=1019.097,-129.008,-94.467,165.327,52.436,159.301
C00862=1019.101,-128.759,-94.476,165.330,52.433,159.302
C00863=1019.105,-128.509,-94.485,165.332,52.431,159.302
C00864=1019.109,-128.260,-94.493,165.335,52.427,159.302
C00865=1019.114,-128.010,-94.501,165.339,52.422,159.302
C00866=1019.119,-127.761,-94.509,165.341,52.418,159.301
C00867=1019.125,-127.511,-94.516,165.344,52.414,159.301
C00868=1019.129,-127.261,-94.523,165.347,52.409,159.301
C00869=1019.135,-127.011,-94.531,165.350,52.405,159.301
C00870=1019.140,-126.762,-94.539,165.353,52.400,159.301
C00871=1019.145,-126.512,-94.546,165.356,52.396,159.300
C00872=1019.150,-126.262,-94.554,165.359,52.391,159.300
C00873=1019.156,-126.012,-94.561,165.362,52.387,159.300
C00874=1019.160,-125.762,-94.568,165.366,52.382,159.300
C00875=1019.166,-125.513,-94.576,165.368,52.378,159.300
C00876=1019.171,-125.262,-94.584,165.372,52.373,159.300
C00877=1019.177,-125.012,-94.591,165.374,52.369,159.299
C00878=1019.181,-124.763,-94.599,165.378,52.365,159.299
C00879=1019.187,-124.513,-94.606,165.380,52.360,159.299
C00880=1019.192,-124.263,-94.614,165.384,52.356,159.299
C00881=1019.196,-124.013,-94.622,165.386,52.351,159.299
C00882=1019.202,-123.764,-94.629,165.389,52.347,159.298
C00883=1019.207,-123.514,-94.637,165.393,52.342,159.298
C00884=1019.212,-123.263,-94.645,165.395,52.338,159.298
C00885=1019.218,-123.015,-94.653,165.399,52.333,159.298
C00886=1019.223,-122.764,-94.660,165.401,52.329,159.298
C00887=1019.228,-122.514,-94.668,165.405,52.325,159.298
C00888=1019.234,-122.265,-94.676,165.407,52.320,159.297
C00889=1019.238,-122.015,-94.683,165.411,52.316,159.297
C00890=1019.243,-121.765,-94.691,165.413,52.311,159.297
C00891=1019.249,-121.515,-94.699,165.416,52.307,159.297
C00892=1019.254,-121.265,-94.707,165.419,52.302,159.297
C00893=1019.259,-121.016,-94.715,165.422,52.298,159.296
C00894=1019.264,-120.766,-94.722,165.426,52.294,159.296
C00895=1019.269,-120.516,-94.731,165.428,52.289,159.296
C00896=1019.274,-120.266,-94.738,165.432,52.285,159.296
C00897=1019.280,-120.016,-94.746,165.434,52.280,159.296
C00898=1019.285,-119.767,-94.754,165.438,52.276,159.296
C00899=1019.290,-119.517,-94.762,165.440,52.271,159.295
C00900=1019.295,-119.267,-94.770,165.444,52.267,159.295
C00901=1019.301,-119.017,-94.778,165.446,52.263,159.295
C00902=1019.306,-118.767,-94.786,165.450,52.258,159.295
C00903=1019.311,-118.517,-94.794,165.453,52.254,159.295
C00904=1019.317,-118.267,-94.801,165.455,52.249,159.294
C00905=1019.323,-117.983,-94.810,165.459,52.244,159.294
C00906=1019.328,-117.699,-94.820,165.463,52.239,159.294
C00907=1019.335,-117.415,-94.828,165.466,52.234,159.294
C00908=1019.340,-117.131,-94.837,165.470,52.229,159.294
C00909=1019.346,-116.881,-94.846,165.472,52.225,159.293
C00910=1019.351,-116.631,-94.854,165.476,52.220,159.293
C00911=1019.357,-116.381,-94.861,165.478,52.216,159.293
C00912=1019.361,-116.132,-94.870,165.482,52.211,159.293
C00913=1019.366,-115.882,-94.877,165.484,52.206,159.292
C00914=1019.371,-115.632,-94.886,165.487,52.202,159.292
C00915=1019.377,-115.383,-94.894,165.490,52.197,159.292
C00916=1019.382,-115.133,-94.902,165.494,52.193,159.292
C00917=1019.388,-114.883,-94.910,165.496,52.188,159.292
C00918=1019.393,-114.633,-94.918,165.500,52.184,159.292
C00919=1019.398,-114.383,-94.926,165.502,52.180,159.291
C00920=1019.403,-114.133,-94.935,165.506,52.175,159.291
C00921=1019.409,-113.884,-94.943,165.508,52.171,159.291
C00922=1019.414,-113.633,-94.950,165.512,52.166,159.291
C00923=1019.419,-113.384,-94.959,165.514,52.162,159.291
C00924=1019.425,-113.134,-94.967,165.517,52.158,159.290
C00925=1019.430,-112.884,-94.976,165.521,52.153,159.290
C00926=1019.435,-112.634,-94.984,165.523,52.149,159.290
C00927=1019.440,-112.384,-94.992,165.527,52.144,159.290
C00928=1019.445,-112.135,-95.001,165.529,52.140,159.290
C00929=1019.451,-111.885,-95.009,165.533,52.135,159.289
C00930=1019.456,-111.635,-95.018,165.535,52.131,159.289
C00931=1019.462,-111.385,-95.025,165.539,52.126,159.289
C00932=1019.467,-111.135,-95.033,165.542,52.122,159.289
C00933=1019.472,-110.886,-95.042,165.545,52.117,159.289
C00934=1019.477,-110.636,-95.050,165.548,52.113,159.288
C00935=1019.483,-110.386,-95.059,165.551,52.109,159.288
C00936=1019.488,-110.137,-95.067,165.554,52.104,159.288
C00937=1019.493,-109.886,-95.075,165.557,52.100,159.288
C00938=1019.498,-109.636,-95.083,165.560,52.095,159.288
C00939=1019.503,-109.387,-95.092,165.563,52.091,159.288
C00940=1019.509,-109.137,-95.100,165.566,52.087,159.287
C00941=1019.515,-108.888,-95.108,165.570,52.082,159.287
C00942=1019.520,-108.638,-95.117,165.572,52.078,159.287
C00943=1019.525,-108.388,-95.125,165.576,52.073,159.287
C00944=1019.530,-108.138,-95.134,165.578,52.068,159.286
C00945=1019.536,-107.889,-95.142,165.581,52.063,159.286
C00946=1019.541,-107.639,-95.151,165.584,52.059,159.286
C00947=1019.546,-107.389,-95.158,165.588,52.055,159.286
C00948=1019.552,-107.138,-95.167,165.590,52.050,159.286
C00949=1019.557,-106.889,-95.176,165.594,52.046,159.286
C00950=1019.562,-106.639,-95.184,165.596,52.042,159.285
C00951=1019.568,-106.390,-95.193,165.600,52.037,159.285
C00952=1019.573,-106.140,-95.202,165.602,52.033,159.285
C00953=1019.578,-105.890,-95.210,165.606,52.028,159.285
C00954=1019.583,-105.640,-95.220,165.609,52.024,159.285
C00955=1019.588,-105.391,-95.228,165.612,52.019,159.284
C00956=1019.593,-105.141,-95.237,165.615,52.015,159.284
C00957=1019.599,-104.890,-95.245,165.618,52.010,159.284
C00958=1019.605,-104.641,-95.254,165.621,52.006,159.284
C00959=1019.610,-104.391,-95.262,165.624,52.001,159.284
C00960=1019.615,-104.141,-95.271,165.627,51.997,159.283
C00961=1019.620,-103.892,-95.279,165.631,51.993,159.283
C00962=1019.626,-103.642,-95.288,165.633,51.988,159.283
C00963=1019.632,-103.392,-95.297,165.636,51.984,159.283
C00964=1019.637,-103.142,-95.306,165.639,51.980,159.283
C00965=1019.642,-102.892,-95.315,165.642,51.975,159.282
C00966=1019.647,-102.643,-95.323,165.645,51.971,159.282
C00967=1019.652,-102.393,-95.332,165.648,51.966,159.282
C00968=1019.658,-102.142,-95.341,165.651,51.962,159.282
C00969=1019.664,-101.859,-95.351,165.655,51.957,159.282
C00970=1019.671,-101.575,-95.361,165.658,51.952,159.281
C00971=1019.677,-101.291,-95.371,165.661,51.947,159.281
C00972=1019.682,-101.006,-95.381,165.665,51.941,159.281
C00973=1019.688,-100.757,-95.390,165.668,51.937,159.281
C00974=1019.693,-100.507,-95.399,165.671,51.933,159.280
C00975=1019.699,-100.257,-95.407,165.674,51.928,159.280
C00976=1019.704,-100.007,-95.416,165.677,51.924,159.280
C00977=1019.710,-99.758,-95.425,165.681,51.919,159.280
C00978=1019.715,-99.508,-95.434,165.684,51.915,159.280
C00979=1019.721,-99.258,-95.442,165.687,51.910,159.279
C00980=1019.725,-99.008,-95.452,165.690,51.906,159.279
C00981=1019.731,-98.759,-95.461,165.692,51.901,159.279
C00982=1019.736,-98.509,-95.469,165.696,51.896,159.279
C00983=1019.742,-98.259,-95.478,165.699,51.892,159.278
C00984=1019.747,-98.009,-95.487,165.702,51.887,159.278
C00985=1019.753,-97.760,-95.496,165.705,51.883,159.278
C00986=1019.758,-97.509,-95.505,165.708,51.878,159.278
C00987=1019.763,-97.260,-95.514,165.711,51.874,159.278
C00988=1019.768,-97.010,-95.524,165.713,51.870,159.277
C00989=1019.774,-96.760,-95.533,165.717,51.865,159.277
C00990=1019.779,-96.510,-95.542,165.720,51.861,159.277
C00991=1019.784,-96.261,-95.551,165.723,51.857,159.277
C00992=1019.790,-96.011,-95.560,165.726,51.852,159.277
C00993=1019.795,-95.761,-95.570,165.729,51.848,159.276
C00994=1019.800,-95.511,-95.578,165.732,51.844,159.276
C00995=1019.806,-95.261,-95.589,165.735,51.839,159.276
C00996=1019.811,-95.012,-95.597,165.738,51.835,159.276
C00997=1019.816,-94.763,-95.606,165.741,51.830,159.276
C00998=1019.822,-94.512,-95.616,165.744,51.826,159.275
C00999=1019.827,-94.263,-95.625,165.747,51.822,159.275
C01000=1019.832,-94.012,-95.634,165.751,51.818,159.275
C01001=1019.838,-93.763,-95.644,165.753,51.814,159.275
C01002=1019.842,-93.513,-95.653,165.757,51.809,159.275
C01003=1019.849,-93.263,-95.662,165.759,51.804,159.274
C01004=1019.854,-93.014,-95.671,165.763,51.799,159.274
C01005=1019.859,-92.763,-95.681,165.765,51.795,159.274
C01006=1019.865,-92.514,-95.690,165.769,51.791,159.274
C01007=1019.869,-92.264,-95.699,165.771,51.786,159.274
C01008=1019.876,-92.014,-95.709,165.775,51.782,159.273
C01009=1019.881,-91.765,-95.718,165.778,51.778,159.273
C01010=1019.886,-91.514,-95.727,165.780,51.773,159.273
C01011=1019.892,-91.265,-95.737,165.784,51.769,159.273
C01012=1019.897,-91.015,-95.747,165.786,51.765,159.273
C01013=1019.903,-90.766,-95.755,165.790,51.760,159.272
C01014=1019.907,-90.516,-95.765,165.792,51.756,159.272
C01015=1019.914,-90.266,-95.775,165.796,51.751,159.272
C01016=1019.918,-90.016,-95.784,165.799,51.747,159.272
C01017=1019.924,-89.767,-95.793,165.802,51.742,159.272
C01018=1019.930,-89.517,-95.802,165.805,51.738,159.271
C01019=1019.935,-89.267,-95.812,165.808,51.734,159.271
C01020=1019.940,-89.018,-95.821,165.811,51.729,159.271
C01021=1019.946,-88.767,-95.831,165.814,51.724,159.271
C01022=1019.951,-88.518,-95.840,165.817,51.720,159.270
C01023=1019.957,-88.268,-95.850,165.820,51.715,159.270
C01024=1019.962,-88.019,-95.859,165.823,51.711,159.270
C01025=1019.968,-87.768,-95.869,165.826,51.707,159.270
C01026=1019.973,-87.519,-95.878,165.829,51.702,159.269
C01027=1019.979,-87.269,-95.887,165.833,51.698,159.269
C01028=1019.984,-87.020,-95.897,165.835,51.694,159.269
C01029=1019.990,-86.770,-95.907,165.838,51.688,159.269
C01030=1019.995,-86.520,-95.917,165.841,51.684,159.268
C01031=1020.001,-86.271,-95.926,165.845,51.680,159.268
C01032=1020.006,-86.020,-95.936,165.848,51.675,159.268
C01033=1020.012,-85.738,-95.946,165.851,51.670,159.268
C01034=1020.019,-85.456,-95.957,165.855,51.665,159.268
C01035=1020.025,-85.174,-95.967,165.858,51.660,159.267
C01036=1020.031,-84.893,-95.978,165.861,51.655,159.267
C01037=1020.037,-84.642,-95.989,165.864,51.650,159.267
C01038=1020.043,-84.393,-95.998,165.868,51.646,159.267
C01039=1020.048,-84.143,-96.008,165.871,51.641,159.266
C01040=1020.054,-83.893,-96.017,165.873,51.636,159.266
C01041=1020.060,-83.643,-96.026,165.877,51.632,159.266
C01042=1020.064,-83.394,-96.036,165.879,51.628,159.266
C01043=1020.071,-83.144,-96.046,165.883,51.623,159.265
C01044=1020.075,-82.894,-96.055,165.886,51.619,159.265
C01045=1020.082,-82.645,-96.065,165.889,51.614,159.265
C01046=1020.087,-82.394,-96.075,165.891,51.609,159.265
C01047=1020.093,-82.145,-96.084,165.895,51.605,159.264
C01048=1020.098,-81.895,-96.095,165.898,51.601,159.264
C01049=1020.104,-81.645,-96.104,165.901,51.595,159.264
C01050=1020.109,-81.396,-96.114,165.904,51.591,159.264
C01051=1020.115,-81.146,-96.124,165.907,51.587,159.263
C01052=1020.121,-80.896,-96.134,165.911,51.582,159.263
C01053=1020.126,-80.647,-96.143,165.913,51.577,159.263
C01054=1020.132,-80.397,-96.153,165.916,51.572,159.263
C01055=1020.138,-80.147,-96.163,165.919,51.568,159.262
C01056=1020.143,-79.897,-96.173,165.923,51.564,159.262
C01057=1020.148,-79.648,-96.183,165.925,51.560,159.262
C01058=1020.154,-79.398,-96.192,165.929,51.555,159.262
C01059=1020.160,-79.148,-96.202,165.931,51.551,159.262
C01060=1020.165,-78.898,-96.212,165.935,51.546,159.261
C01061=1020.170,-78.648,-96.222,165.938,51.542,159.261
C01062=1020.176,-78.399,-96.233,165.941,51.537,159.261
C01063=1020.182,-78.149,-96.243,165.943,51.533,159.261
C01064=1020.187,-77.900,-96.252,165.947,51.528,159.260
C01065=1020.192,-77.649,-96.263,165.950,51.524,159.260
C01066=1020.198,-77.400,-96.272,165.952,51.520,159.260
C01067=1020.203,-77.151,-96.283,165.956,51.515,159.260
C01068=1020.209,-76.901,-96.293,165.958,51.511,159.259
C01069=1020.214,-76.651,-96.303,165.962,51.506,159.259
C01070=1020.220,-76.401,-96.313,165.964,51.501,159.259
C01071=1020.226,-76.151,-96.323,165.968,51.497,159.259
C01072=1020.231,-75.902,-96.333,165.970,51.493,159.258
C01073=1020.236,-75.652,-96.343,165.974,51.488,159.258
C01074=1020.243,-75.402,-96.353,165.976,51.484,159.258
C01075=1020.248,-75.152,-96.363,165.980,51.479,159.258
C01076=1020.253,-74.903,-96.374,165.983,51.475,159.258
C01077=1020.259,-74.653,-96.384,165.986,51.470,159.257
C01078=1020.265,-74.403,-96.393,165.988,51.466,159.257
C01079=1020.270,-74.153,-96.405,165.992,51.461,159.257
C01080=1020.275,-73.903,-96.415,165.995,51.457,159.256
C01081=1020.281,-73.653,-96.425,165.998,51.452,159.256
C01082=1020.286,-73.404,-96.436,166.001,51.448,159.256
C01083=1020.291,-73.154,-96.446,166.003,51.444,159.256
C01084=1020.297,-72.905,-96.457,166.007,51.440,159.256
C01085=1020.302,-72.655,-96.467,166.010,51.435,159.255
C01086=1020.308,-72.405,-96.478,166.012,51.431,159.255
C01087=1020.314,-72.155,-96.488,166.016,51.427,159.255
C01088=1020.319,-71.906,-96.498,166.018,51.422,159.255
C01089=1020.324,-71.656,-96.509,166.022,51.418,159.254
C01090=1020.330,-71.407,-96.520,166.025,51.414,159.254
C01091=1020.335,-71.157,-96.530,166.028,51.409,159.254
C01092=1020.341,-70.907,-96.541,166.031,51.405,159.254
C01093=1020.347,-70.657,-96.551,166.033,51.401,159.253
C01094=1020.352,-70.407,-96.562,166.037,51.396,159.253
C01095=1020.357,-70.158,-96.571,166.040,51.392,159.253
C01096=1020.363,-69.909,-96.582,166.043,51.388,159.253
C01097=1020.369,-69.628,-96.594,166.047,51.383,159.253
C01098=1020.375,-69.348,-96.606,166.049,51.378,159.252
C01099=1020.381,-69.068,-96.618,166.053,51.374,159.252
C01100=1020.387,-68.788,-96.630,166.056,51.368,159.252
C01101=1020.393,-68.538,-96.641,166.059,51.364,159.252
C01102=1020.399,-68.289,-96.651,166.062,51.360,159.251
C01103=1020.404,-68.038,-96.662,166.066,51.355,159.251
C01104=1020.410,-67.789,-96.672,166.068,51.351,159.251
C01105=1020.414,-67.540,-96.684,166.072,51.346,159.251
C01106=1020.420,-67.290,-96.694,166.074,51.342,159.250
C01107=1020.426,-67.040,-96.705,166.077,51.337,159.250
C01108=1020.431,-66.790,-96.715,166.080,51.333,159.250
C01109=1020.437,-66.541,-96.726,166.083,51.329,159.250
C01110=1020.443,-66.291,-96.736,166.087,51.324,159.249
C01111=1020.448,-66.041,-96.747,166.089,51.320,159.249
C01112=1020.454,-65.792,-96.758,166.093,51.315,159.249
C01113=1020.459,-65.542,-96.768,166.095,51.311,159.249
C01114=1020.465,-65.292,-96.779,166.098,51.307,159.248
C01115=1020.471,-65.042,-96.789,166.101,51.302,159.248
C01116=1020.476,-64.793,-96.800,166.104,51.298,159.248
C01117=1020.482,-64.544,-96.811,166.107,51.293,159.248
C01118=1020.487,-64.293,-96.822,166.110,51.289,159.247
C01119=1020.493,-64.044,-96.833,166.114,51.284,159.247
C01120=1020.498,-63.794,-96.844,166.116,51.280,159.247
C01121=1020.504,-63.545,-96.855,166.119,51.275,159.247
C01122=1020.509,-63.295,-96.865,166.122,51.271,159.246
C01123=1020.515,-63.045,-96.876,166.126,51.266,159.246
C01124=1020.522,-62.795,-96.887,166.128,51.262,159.246
C01125=1020.527,-62.545,-96.898,166.131,51.258,159.246
C01126=1020.533,-62.295,-96.908,166.134,51.253,159.245
C01127=1020.538,-62.046,-96.919,166.137,51.249,159.245
C01128=1020.543,-61.796,-96.930,166.140,51.244,159.245
C01129=1020.549,-61.546,-96.941,166.143,51.240,159.244
C01130=1020.555,-61.297,-96.952,166.146,51.235,159.244
C01131=1020.560,-61.047,-96.962,166.149,51.230,159.244
C01132=1020.566,-60.797,-96.973,166.152,51.226,159.244
C01133=1020.572,-60.548,-96.984,166.155,51.222,159.243
C01134=1020.578,-60.298,-96.995,166.159,51.217,159.243
C01135=1020.583,-60.049,-97.006,166.161,51.212,159.243
C01136=1020.590,-59.799,-97.017,166.164,51.208,159.243
C01137=1020.595,-59.549,-97.028,166.167,51.204,159.242
C01138=1020.600,-59.299,-97.039,166.171,51.199,159.242
C01139=1020.606,-59.049,-97.049,166.173,51.194,159.242
C01140=1020.612,-58.800,-97.060,166.176,51.190,159.241
C01141=1020.617,-58.550,-97.071,166.179,51.186,159.241
C01142=1020.623,-58.301,-97.082,166.183,51.181,159.241
C01143=1020.629,-58.051,-97.093,166.185,51.176,159.241
///RCONF 1,0,0,0,0,0,0,0,0,0,0,0,0,0,0,0,0,0,0,0,0,0,0,0
C01144=1020.635,-57.801,-97.104,166.187,51.172,159.240
C01145=1020.641,-57.552,-97.115,166.191,51.168,159.240
C01146=1020.646,-57.302,-97.127,166.193,51.163,159.240
C01147=1020.652,-57.052,-97.137,166.197,51.158,159.239
C01148=1020.657,-56.803,-97.148,166.199,51.154,159.239
C01149=1020.664,-56.553,-97.160,166.203,51.149,159.239
C01150=1020.669,-56.303,-97.170,166.205,51.145,159.238
C01151=1020.675,-56.054,-97.181,166.209,51.140,159.238
C01152=1020.681,-55.804,-97.192,166.211,51.135,159.238
C01153=1020.687,-55.554,-97.203,166.215,51.131,159.238
C01154=1020.692,-55.304,-97.215,166.217,51.127,159.237
C01155=1020.698,-55.055,-97.226,166.221,51.121,159.237
C01156=1020.704,-54.805,-97.237,166.223,51.117,159.237
C01157=1020.709,-54.556,-97.248,166.227,51.113,159.237
C01158=1020.716,-54.306,-97.259,166.229,51.108,159.236
C01159=1020.722,-54.056,-97.270,166.233,51.103,159.236
C01160=1020.727,-53.807,-97.281,166.235,51.099,159.236
C01161=1020.734,-53.528,-97.293,166.240,51.094,159.235
C01162=1020.740,-53.248,-97.305,166.243,51.089,159.235
C01163=1020.747,-52.969,-97.317,166.246,51.083,159.235
C01164=1020.753,-52.690,-97.330,166.249,51.078,159.234
C01165=1020.759,-52.441,-97.341,166.252,51.073,159.234
C01166=1020.765,-52.191,-97.352,166.255,51.069,159.234
C01167=1020.771,-51.942,-97.364,166.258,51.065,159.233
C01168=1020.777,-51.692,-97.375,166.261,51.059,159.233
C01169=1020.782,-51.443,-97.386,166.264,51.055,159.233
C01170=1020.788,-51.192,-97.397,166.267,51.050,159.232
C01171=1020.794,-50.943,-97.408,166.270,51.046,159.232
C01172=1020.800,-50.693,-97.420,166.273,51.041,159.232
C01173=1020.805,-50.444,-97.432,166.276,51.037,159.232
C01174=1020.811,-50.194,-97.443,166.278,51.032,159.231
C01175=1020.816,-49.944,-97.454,166.282,51.028,159.231
C01176=1020.822,-49.694,-97.467,166.284,51.024,159.231
C01177=1020.828,-49.445,-97.478,166.288,51.019,159.230
C01178=1020.833,-49.195,-97.489,166.290,51.015,159.230
C01179=1020.840,-48.945,-97.501,166.293,51.011,159.230
C01180=1020.845,-48.696,-97.512,166.296,51.006,159.230
C01181=1020.850,-48.446,-97.523,166.299,51.002,159.229
C01182=1020.856,-48.196,-97.536,166.303,50.997,159.229
C01183=1020.862,-47.947,-97.547,166.305,50.993,159.229
C01184=1020.867,-47.697,-97.558,166.308,50.989,159.228
C01185=1020.874,-47.447,-97.570,166.311,50.984,159.228
C01186=1020.879,-47.198,-97.582,166.314,50.980,159.228
C01187=1020.885,-46.948,-97.594,166.316,50.975,159.228
C01188=1020.890,-46.698,-97.605,166.320,50.971,159.227
C01189=1020.896,-46.449,-97.617,166.323,50.967,159.227
C01190=1020.902,-46.199,-97.629,166.326,50.962,159.227
C01191=1020.907,-45.949,-97.640,166.328,50.957,159.226
C01192=1020.913,-45.700,-97.652,166.331,50.953,159.226
C01193=1020.919,-45.450,-97.663,166.335,50.949,159.226
C01194=1020.925,-45.201,-97.675,166.337,50.944,159.225
C01195=1020.930,-44.950,-97.687,166.341,50.939,159.225
C01196=1020.936,-44.701,-97.698,166.343,50.935,159.225
C01197=1020.942,-44.451,-97.710,166.346,50.930,159.225
C01198=1020.948,-44.202,-97.722,166.349,50.926,159.224
C01199=1020.953,-43.952,-97.733,166.352,50.922,159.224
C01200=1020.959,-43.702,-97.746,166.355,50.917,159.224
C01201=1020.964,-43.453,-97.757,166.357,50.913,159.223
C01202=1020.970,-43.203,-97.769,166.361,50.908,159.223
C01203=1020.976,-42.954,-97.780,166.364,50.904,159.223
C01204=1020.982,-42.704,-97.793,166.366,50.899,159.222
C01205=1020.988,-42.454,-97.804,166.370,50.895,159.222
C01206=1020.994,-42.204,-97.816,166.372,50.890,159.222
C01207=1021.000,-41.955,-97.828,166.375,50.885,159.222
C01208=1021.005,-41.705,-97.840,166.378,50.881,159.221
C01209=1021.011,-41.456,-97.852,166.382,50.877,159.221
C01210=1021.017,-41.206,-97.863,166.384,50.872,159.221
C01211=1021.022,-40.956,-97.875,166.387,50.868,159.220
C01212=1021.029,-40.707,-97.887,166.390,50.863,159.220
C01213=1021.034,-40.457,-97.899,166.392,50.858,159.220
C01214=1021.041,-40.207,-97.911,166.396,50.854,159.219
C01215=1021.046,-39.958,-97.922,166.399,50.850,159.219
C01216=1021.052,-39.708,-97.935,166.402,50.845,159.219
C01217=1021.058,-39.459,-97.946,166.405,50.840,159.219
C01218=1021.063,-39.208,-97.958,166.407,50.836,159.218
C01219=1021.068,-38.959,-97.970,166.410,50.831,159.218
C01220=1021.074,-38.709,-97.983,166.413,50.827,159.218
C01221=1021.080,-38.460,-97.994,166.416,50.823,159.217
C01222=1021.086,-38.210,-98.006,166.419,50.818,159.217
C01223=1021.092,-37.960,-98.019,166.422,50.814,159.217
C01224=1021.097,-37.711,-98.031,166.424,50.809,159.216
C01225=1021.104,-37.433,-98.044,166.428,50.805,159.216
C01226=1021.110,-37.154,-98.058,166.431,50.800,159.216
C01227=1021.116,-36.876,-98.072,166.434,50.795,159.215
C01228=1021.123,-36.597,-98.085,166.438,50.790,159.215
C01229=1021.129,-36.347,-98.097,166.440,50.785,159.215
C01230=1021.134,-36.097,-98.110,166.444,50.781,159.215
C01231=1021.140,-35.848,-98.122,166.447,50.777,159.214
C01232=1021.146,-35.598,-98.134,166.449,50.772,159.214
C01233=1021.152,-35.349,-98.146,166.452,50.768,159.214
C01234=1021.158,-35.099,-98.159,166.455,50.763,159.213
C01235=1021.164,-34.849,-98.171,166.457,50.759,159.213
C01236=1021.169,-34.599,-98.183,166.461,50.754,159.213
C01237=1021.174,-34.349,-98.195,166.464,50.750,159.212
C01238=1021.180,-34.100,-98.207,166.466,50.746,159.212
C01239=1021.186,-33.851,-98.219,166.470,50.741,159.212
C01240=1021.192,-33.601,-98.232,166.472,50.737,159.211
C01241=1021.198,-33.352,-98.244,166.476,50.732,159.211
C01242=1021.203,-33.102,-98.257,166.478,50.727,159.211
C01243=1021.209,-32.852,-98.269,166.481,50.723,159.210
C01244=1021.215,-32.603,-98.281,166.484,50.719,159.210
C01245=1021.221,-32.353,-98.293,166.487,50.714,159.210
C01246=1021.227,-32.103,-98.306,166.489,50.710,159.209
C01247=1021.233,-31.854,-98.318,166.493,50.705,159.209
C01248=1021.238,-31.604,-98.331,166.495,50.700,159.209
C01249=1021.244,-31.354,-98.343,166.499,50.696,159.208
C01250=1021.250,-31.105,-98.355,166.501,50.692,159.208
C01251=1021.256,-30.855,-98.368,166.504,50.687,159.208
C01252=1021.262,-30.605,-98.381,166.507,50.683,159.208
C01253=1021.268,-30.356,-98.392,166.510,50.678,159.207
C01254=1021.273,-30.107,-98.405,166.512,50.674,159.207
C01255=1021.279,-29.857,-98.417,166.516,50.669,159.207
C01256=1021.285,-29.607,-98.430,166.518,50.664,159.206
C01257=1021.291,-29.358,-98.442,166.522,50.660,159.206
C01258=1021.296,-29.108,-98.455,166.524,50.655,159.205
C01259=1021.302,-28.858,-98.467,166.527,50.651,159.205
C01260=1021.309,-28.608,-98.479,166.530,50.647,159.205
C01261=1021.314,-28.359,-98.491,166.533,50.642,159.204
C01262=1021.320,-28.109,-98.504,166.536,50.637,159.204
C01263=1021.326,-27.859,-98.516,166.538,50.633,159.204
C01264=1021.332,-27.609,-98.529,166.541,50.628,159.203
C01265=1021.338,-27.361,-98.542,166.545,50.624,159.203
C01266=1021.344,-27.111,-98.554,166.547,50.619,159.203
C01267=1021.350,-26.861,-98.567,166.550,50.615,159.202
C01268=1021.355,-26.611,-98.580,166.553,50.611,159.202
C01269=1021.361,-26.361,-98.593,166.556,50.606,159.202
C01270=1021.366,-26.112,-98.606,166.558,50.602,159.201
C01271=1021.372,-25.863,-98.618,166.561,50.598,159.201
C01272=1021.378,-25.613,-98.631,166.564,50.593,159.201
C01273=1021.384,-25.363,-98.643,166.567,50.588,159.200
C01274=1021.390,-25.114,-98.656,166.569,50.584,159.200
C01275=1021.395,-24.864,-98.669,166.573,50.580,159.200
C01276=1021.401,-24.614,-98.682,166.575,50.575,159.199
C01277=1021.407,-24.365,-98.695,166.578,50.571,159.199
C01278=1021.413,-24.115,-98.708,166.582,50.566,159.199
C01279=1021.419,-23.865,-98.720,166.584,50.562,159.199
C01280=1021.424,-23.616,-98.732,166.586,50.558,159.198
C01281=1021.430,-23.367,-98.746,166.589,50.553,159.198
C01282=1021.435,-23.116,-98.759,166.593,50.549,159.198
C01283=1021.441,-22.867,-98.771,166.595,50.544,159.197
C01284=1021.447,-22.617,-98.785,166.598,50.540,159.197
C01285=1021.453,-22.367,-98.797,166.601,50.535,159.196
C01286=1021.459,-22.119,-98.810,166.604,50.531,159.196
C01287=1021.465,-21.869,-98.823,166.606,50.527,159.196
C01288=1021.471,-21.619,-98.835,166.609,50.522,159.195
C01289=1021.477,-21.340,-98.850,166.613,50.516,159.195
C01290=1021.484,-21.060,-98.864,166.615,50.512,159.195
C01291=1021.490,-20.781,-98.878,166.619,50.507,159.194
C01292=1021.497,-20.502,-98.893,166.622,50.502,159.194
C01293=1021.502,-20.252,-98.907,166.624,50.497,159.194
C01294=1021.508,-20.002,-98.919,166.628,50.493,159.193
C01295=1021.514,-19.753,-98.932,166.631,50.489,159.193
C01296=1021.520,-19.503,-98.945,166.633,50.484,159.193
C01297=1021.526,-19.254,-98.958,166.637,50.480,159.192
C01298=1021.532,-19.004,-98.971,166.639,50.475,159.192
C01299=1021.537,-18.754,-98.984,166.641,50.471,159.192
C01300=1021.544,-18.504,-98.997,166.645,50.466,159.191
C01301=1021.549,-18.271,-99.010,166.647,50.461,159.191
C01302=1021.555,-18.038,-99.021,166.650,50.457,159.191
C01303=1021.560,-17.805,-99.033,166.653,50.453,159.190
C01304=1021.566,-17.571,-99.046,166.655,50.449,159.190
C01305=1021.571,-17.337,-99.057,166.658,50.445,159.190
C01306=1021.576,-17.104,-99.070,166.660,50.440,159.189
C01307=1021.582,-16.870,-99.082,166.663,50.436,159.189
C01308=1021.587,-16.637,-99.094,166.665,50.432,159.188
C01309=1021.594,-16.388,-99.108,166.669,50.428,159.188
C01310=1021.600,-16.138,-99.120,166.671,50.423,159.188
C01311=1021.606,-15.888,-99.133,166.674,50.419,159.187
C01312=1021.611,-15.638,-99.147,166.676,50.414,159.187
C01313=1021.617,-15.389,-99.160,166.680,50.410,159.187
C01314=1021.623,-15.140,-99.173,166.683,50.406,159.186
C01315=1021.629,-14.890,-99.186,166.685,50.401,159.186
C01316=1021.635,-14.640,-99.199,166.688,50.397,159.186
C01317=1021.640,-14.391,-99.213,166.691,50.392,159.185
C01318=1021.646,-14.141,-99.227,166.693,50.387,159.185
C01319=1021.652,-13.891,-99.240,166.696,50.383,159.185
C01320=1021.658,-13.642,-99.253,166.700,50.379,159.184
C01321=1021.663,-13.392,-99.267,166.702,50.374,159.184
C01322=1021.669,-13.143,-99.279,166.705,50.370,159.184
C01323=1021.675,-12.893,-99.293,166.707,50.365,159.183
C01324=1021.681,-12.644,-99.307,166.711,50.361,159.183
C01325=1021.687,-12.394,-99.320,166.713,50.357,159.183
C01326=1021.692,-12.144,-99.333,166.716,50.352,159.182
C01327=1021.699,-11.895,-99.346,166.718,50.348,159.182
C01328=1021.704,-11.645,-99.360,166.722,50.343,159.182
C01329=1021.710,-11.396,-99.373,166.724,50.339,159.181
C01330=1021.715,-11.146,-99.387,166.727,50.335,159.181
C01331=1021.722,-10.897,-99.400,166.729,50.330,159.180
C01332=1021.728,-10.647,-99.413,166.733,50.325,159.180
C01333=1021.733,-10.398,-99.427,166.735,50.321,159.180
C01334=1021.739,-10.149,-99.440,166.738,50.317,159.179
C01335=1021.745,-9.899,-99.454,166.741,50.312,159.179
C01336=1021.751,-9.649,-99.467,166.744,50.307,159.179
C01337=1021.757,-9.399,-99.481,166.746,50.303,159.178
C01338=1021.763,-9.150,-99.494,166.749,50.299,159.178
C01339=1021.769,-8.900,-99.508,166.752,50.294,159.178
C01340=1021.775,-8.651,-99.521,166.755,50.289,159.177
C01341=1021.780,-8.401,-99.535,166.757,50.285,159.177
C01342=1021.786,-8.151,-99.548,166.761,50.280,159.176
C01343=1021.792,-7.902,-99.562,166.763,50.276,159.176
C01344=1021.798,-7.652,-99.575,166.766,50.272,159.176
C01345=1021.803,-7.403,-99.589,166.768,50.267,159.175
C01346=1021.810,-7.153,-99.602,166.772,50.263,159.175
C01347=1021.816,-6.904,-99.616,166.774,50.258,159.175
C01348=1021.822,-6.654,-99.629,166.777,50.254,159.174
C01349=1021.828,-6.405,-99.643,166.780,50.249,159.174
C01350=1021.834,-6.155,-99.657,166.783,50.245,159.174
C01351=1021.840,-5.906,-99.670,166.785,50.240,159.173
C01352=1021.845,-5.656,-99.684,166.787,50.235,159.172
C01353=1021.853,-5.342,-99.700,166.792,50.230,159.172
C01354=1021.860,-5.029,-99.717,166.795,50.224,159.172
C01355=1021.868,-4.715,-99.735,166.799,50.218,159.171
C01356=1021.876,-4.402,-99.752,166.802,50.213,159.171
C01357=1021.881,-4.152,-99.766,166.804,50.208,159.170
C01358=1021.887,-3.903,-99.780,166.807,50.204,159.170
C01359=1021.893,-3.654,-99.793,166.810,50.199,159.170
C01360=1021.899,-3.403,-99.807,166.813,50.195,159.169
C01361=1021.904,-3.154,-99.821,166.815,50.191,159.169
C01362=1021.910,-2.904,-99.835,166.818,50.187,159.169
C01363=1021.915,-2.655,-99.849,166.820,50.182,159.168
C01364=1021.921,-2.406,-99.863,166.824,50.178,159.168
C01365=1021.928,-2.156,-99.877,166.826,50.173,159.167
C01366=1021.934,-1.906,-99.891,166.829,50.169,159.167
C01367=1021.939,-1.657,-99.905,166.832,50.165,159.167
C01368=1021.944,-1.407,-99.918,166.834,50.160,159.166
C01369=1021.950,-1.158,-99.933,166.838,50.156,159.166
C01370=1021.956,-0.908,-99.947,166.840,50.151,159.166
C01371=1021.963,-0.658,-99.960,166.843,50.147,159.165
C01372=1021.968,-0.409,-99.974,166.845,50.143,159.165
C01373=1021.974,-0.160,-99.989,166.848,50.139,159.165
C01374=1021.980,0.090,-100.003,166.850,50.134,159.164
C01375=1021.985,0.340,-100.017,166.854,50.129,159.164
C01376=1021.991,0.589,-100.031,166.856,50.125,159.163
C01377=1021.997,0.838,-100.045,166.859,50.121,159.163
C01378=1022.003,1.088,-100.059,166.862,50.117,159.163
C01379=1022.009,1.338,-100.073,166.864,50.112,159.162
C01380=1022.014,1.588,-100.087,166.868,50.107,159.162
C01381=1022.020,1.836,-100.101,166.870,50.103,159.162
C01382=1022.026,2.087,-100.116,166.873,50.099,159.161
C01383=1022.032,2.336,-100.130,166.875,50.094,159.161
C01384=1022.038,2.585,-100.144,166.877,50.090,159.160
C01385=1022.044,2.835,-100.157,166.881,50.085,159.160
C01386=1022.050,3.085,-100.172,166.883,50.081,159.160
C01387=1022.055,3.334,-100.185,166.886,50.077,159.159
C01388=1022.061,3.583,-100.200,166.888,50.072,159.159
C01389=1022.067,3.834,-100.214,166.892,50.067,159.159
C01390=1022.074,4.082,-100.228,166.894,50.063,159.158
C01391=1022.079,4.332,-100.242,166.897,50.059,159.158
C01392=1022.085,4.582,-100.256,166.899,50.054,159.157
C01393=1022.091,4.831,-100.271,166.902,50.050,159.157
C01394=1022.096,5.081,-100.285,166.905,50.045,159.157
C01395=1022.103,5.331,-100.299,166.908,50.041,159.156
C01396=1022.108,5.580,-100.314,166.910,50.036,159.156
C01397=1022.115,5.829,-100.327,166.913,50.032,159.155
C01398=1022.121,6.079,-100.342,166.915,50.027,159.155
C01399=1022.126,6.328,-100.356,166.919,50.023,159.155
C01400=1022.132,6.578,-100.370,166.921,50.018,159.154
C01401=1022.138,6.828,-100.384,166.924,50.014,159.154
C01402=1022.144,7.077,-100.398,166.926,50.009,159.153
C01403=1022.150,7.326,-100.413,166.930,50.004,159.153
C01404=1022.156,7.576,-100.427,166.932,50.000,159.153
C01405=1022.162,7.825,-100.441,166.935,49.995,159.152
C01406=1022.168,8.075,-100.455,166.937,49.991,159.152
C01407=1022.174,8.325,-100.469,166.941,49.986,159.151
C01408=1022.179,8.574,-100.484,166.943,49.982,159.151
C01409=1022.186,8.824,-100.498,166.946,49.978,159.151
C01410=1022.191,9.073,-100.513,166.948,49.973,159.150
C01411=1022.197,9.323,-100.527,166.951,49.969,159.150
C01412=1022.204,9.572,-100.541,166.954,49.964,159.149
C01413=1022.209,9.822,-100.555,166.957,49.960,159.149
C01414=1022.216,10.071,-100.570,166.959,49.955,159.149
C01415=1022.221,10.321,-100.584,166.961,49.950,159.148
C01416=1022.228,10.571,-100.598,166.965,49.946,159.148
C01417=1022.234,10.853,-100.614,166.968,49.941,159.147
C01418=1022.241,11.137,-100.631,166.970,49.935,159.147
C01419=1022.248,11.420,-100.647,166.974,49.930,159.146
C01420=1022.255,11.703,-100.663,166.977,49.925,159.146
C01421=1022.261,11.952,-100.678,166.979,49.920,159.145
C01422=1022.267,12.202,-100.693,166.982,49.916,159.145
C01423=1022.272,12.451,-100.707,166.985,49.911,159.145
C01424=1022.279,12.701,-100.721,166.988,49.907,159.144
C01425=1022.284,12.950,-100.735,166.990,49.903,159.144
C01426=1022.291,13.200,-100.750,166.993,49.898,159.143
C01427=1022.297,13.449,-100.764,166.996,49.893,159.143
C01428=1022.303,13.699,-100.779,166.999,49.889,159.143
C01429=1022.308,13.948,-100.794,167.001,49.884,159.142
C01430=1022.315,14.198,-100.809,167.004,49.880,159.142
C01431=1022.320,14.447,-100.823,167.006,49.875,159.141
C01432=1022.326,14.696,-100.837,167.010,49.871,159.141
C01433=1022.332,14.946,-100.852,167.012,49.866,159.141
C01434=1022.338,15.195,-100.867,167.015,49.862,159.140
C01435=1022.343,15.446,-100.881,167.017,49.857,159.140
C01436=1022.349,15.695,-100.896,167.020,49.853,159.139
C01437=1022.356,15.944,-100.911,167.022,49.849,159.139
C01438=1022.361,16.193,-100.926,167.026,49.844,159.139
C01439=1022.368,16.443,-100.940,167.028,49.840,159.138
C01440=1022.373,16.692,-100.954,167.030,49.835,159.138
C01441=1022.379,16.942,-100.970,167.033,49.831,159.137
C01442=1022.385,17.192,-100.985,167.035,49.826,159.137
C01443=1022.391,17.441,-100.999,167.038,49.822,159.136
C01444=1022.397,17.691,-101.014,167.041,49.817,159.136
C01445=1022.403,17.940,-101.028,167.044,49.813,159.136
C01446=1022.409,18.190,-101.043,167.046,49.808,159.135
C01447=1022.414,18.439,-101.058,167.049,49.804,159.135
C01448=1022.421,18.689,-101.073,167.051,49.800,159.134
C01449=1022.426,18.938,-101.088,167.055,49.794,159.134
C01450=1022.433,19.187,-101.103,167.057,49.790,159.134
C01451=1022.439,19.437,-101.118,167.060,49.786,159.133
C01452=1022.444,19.686,-101.133,167.062,49.782,159.133
C01453=1022.450,19.937,-101.147,167.065,49.777,159.132
C01454=1022.456,20.186,-101.162,167.067,49.773,159.132
C01455=1022.462,20.436,-101.177,167.070,49.768,159.131
C01456=1022.468,20.685,-101.192,167.073,49.763,159.131
C01457=1022.474,20.934,-101.207,167.076,49.759,159.131
C01458=1022.480,21.184,-101.222,167.078,49.754,159.130
C01459=1022.485,21.433,-101.237,167.081,49.750,159.130
C01460=1022.492,21.683,-101.252,167.083,49.746,159.129
C01461=1022.497,21.932,-101.267,167.086,49.742,159.129
C01462=1022.503,22.182,-101.282,167.089,49.737,159.129
C01463=1022.510,22.431,-101.297,167.092,49.733,159.128
C01464=1022.515,22.681,-101.312,167.094,49.728,159.128
C01465=1022.521,22.930,-101.327,167.096,49.723,159.127
C01466=1022.527,23.179,-101.342,167.099,49.719,159.127
C01467=1022.532,23.429,-101.357,167.102,49.714,159.126
C01468=1022.539,23.679,-101.372,167.105,49.710,159.126
C01469=1022.545,23.928,-101.387,167.108,49.705,159.126
C01470=1022.550,24.178,-101.402,167.110,49.701,159.125
C01471=1022.557,24.427,-101.418,167.113,49.697,159.125
C01472=1022.563,24.676,-101.432,167.115,49.692,159.124
C01473=1022.568,24.926,-101.448,167.118,49.688,159.124
C01474=1022.575,25.175,-101.463,167.121,49.683,159.124
C01475=1022.581,25.424,-101.478,167.123,49.678,159.123
C01476=1022.586,25.674,-101.493,167.126,49.674,159.123
C01477=1022.593,25.924,-101.508,167.128,49.670,159.122
C01478=1022.598,26.173,-101.523,167.131,49.665,159.122
C01479=1022.604,26.423,-101.538,167.133,49.661,159.121
C01480=1022.610,26.673,-101.553,167.136,49.656,159.121
C01481=1022.617,26.956,-101.570,167.139,49.651,159.120
C01482=1022.624,27.241,-101.587,167.142,49.646,159.120
C01483=1022.631,27.525,-101.605,167.145,49.640,159.119
C01484=1022.637,27.810,-101.623,167.148,49.636,159.119
C01485=1022.643,28.059,-101.638,167.152,49.631,159.119
C01486=1022.649,28.309,-101.654,167.154,49.627,159.118
C01487=1022.655,28.558,-101.668,167.157,49.623,159.118
C01488=1022.661,28.808,-101.684,167.159,49.618,159.117
C01489=1022.666,29.057,-101.700,167.161,49.613,159.117
C01490=1022.672,29.306,-101.715,167.164,49.609,159.117
C01491=1022.678,29.556,-101.730,167.166,49.605,159.116
C01492=1022.684,29.806,-101.745,167.169,49.601,159.116
C01493=1022.690,30.055,-101.762,167.171,49.596,159.115
C01494=1022.696,30.304,-101.776,167.175,49.592,159.115
C01495=1022.702,30.554,-101.792,167.177,49.587,159.114
C01496=1022.708,30.804,-101.808,167.180,49.582,159.114
C01497=1022.713,31.053,-101.822,167.182,49.578,159.114
C01498=1022.719,31.303,-101.838,167.185,49.573,159.113
C01499=1022.726,31.552,-101.854,167.187,49.569,159.113
C01500=1022.731,31.802,-101.869,167.190,49.565,159.112
C01501=1022.737,32.051,-101.884,167.192,49.560,159.112
C01502=1022.743,32.300,-101.900,167.196,49.556,159.111
C01503=1022.749,32.550,-101.916,167.198,49.551,159.111
C01504=1022.755,32.800,-101.931,167.201,49.547,159.111
C01505=1022.760,33.048,-101.946,167.203,49.542,159.110
C01506=1022.767,33.298,-101.961,167.206,49.538,159.110
C01507=1022.773,33.547,-101.978,167.208,49.534,159.109
C01508=1022.778,33.797,-101.993,167.211,49.529,159.109
C01509=1022.785,34.047,-102.008,167.214,49.524,159.108
C01510=1022.790,34.295,-102.024,167.217,49.520,159.108
C01511=1022.797,34.545,-102.039,167.219,49.515,159.107
C01512=1022.803,34.794,-102.055,167.221,49.511,159.107
C01513=1022.808,35.044,-102.071,167.224,49.507,159.107
C01514=1022.815,35.294,-102.086,167.227,49.502,159.106
C01515=1022.820,35.543,-102.102,167.229,49.497,159.106
C01516=1022.826,35.792,-102.117,167.233,49.493,159.105
C01517=1022.832,36.042,-102.133,167.235,49.488,159.105
C01518=1022.839,36.291,-102.148,167.237,49.483,159.104
C01519=1022.845,36.541,-102.164,167.240,49.479,159.104
C01520=1022.850,36.791,-102.180,167.242,49.475,159.103
C01521=1022.856,37.039,-102.195,167.245,49.470,159.103
C01522=1022.862,37.289,-102.210,167.247,49.466,159.103
C01523=1022.868,37.538,-102.227,167.250,49.461,159.102
C01524=1022.874,37.788,-102.242,167.254,49.457,159.102
C01525=1022.879,38.038,-102.258,167.256,49.452,159.101
C01526=1022.885,38.287,-102.275,167.259,49.448,159.101
C01527=1022.891,38.537,-102.290,167.261,49.444,159.100
C01528=1022.897,38.785,-102.306,167.263,49.439,159.100
C01529=1022.903,39.035,-102.321,167.266,49.435,159.100
C01530=1022.909,39.285,-102.337,167.268,49.430,159.099
C01531=1022.915,39.534,-102.354,167.271,49.426,159.099
C01532=1022.920,39.784,-102.369,167.273,49.422,159.098
C01533=1022.926,40.033,-102.385,167.276,49.417,159.098
C01534=1022.933,40.282,-102.401,167.278,49.413,159.097
C01535=1022.938,40.532,-102.416,167.282,49.408,159.097
C01536=1022.944,40.781,-102.432,167.285,49.404,159.097
C01537=1022.950,41.030,-102.449,167.287,49.399,159.096
C01538=1022.956,41.280,-102.464,167.289,49.395,159.096
C01539=1022.962,41.530,-102.481,167.292,49.391,159.095
C01540=1022.967,41.779,-102.497,167.294,49.386,159.095
C01541=1022.974,42.029,-102.512,167.297,49.381,159.094
C01542=1022.980,42.278,-102.528,167.299,49.377,159.094
C01543=1022.986,42.527,-102.544,167.302,49.373,159.093
C01544=1022.992,42.777,-102.560,167.305,49.369,159.093
C01545=1022.998,43.061,-102.578,167.308,49.363,159.092
C01546=1023.004,43.346,-102.597,167.311,49.358,159.092
C01547=1023.011,43.630,-102.616,167.313,49.353,159.091
C01548=1023.017,43.914,-102.634,167.317,49.349,159.091
C01549=1023.023,44.164,-102.650,167.319,49.345,159.091
C01550=1023.029,44.413,-102.666,167.322,49.340,159.090
C01551=1023.035,44.663,-102.682,167.325,49.336,159.090
C01552=1023.041,44.912,-102.699,167.327,49.331,159.089
C01553=1023.046,45.162,-102.715,167.330,49.327,159.089
C01554=1023.052,45.411,-102.732,167.332,49.323,159.088
C01555=1023.058,45.660,-102.748,167.335,49.319,159.088
C01556=1023.064,45.910,-102.764,167.337,49.314,159.088
C01557=1023.070,46.159,-102.780,167.339,49.309,159.087
C01558=1023.076,46.408,-102.797,167.342,49.305,159.087
C01559=1023.081,46.658,-102.812,167.345,49.301,159.086
C01560=1023.087,46.907,-102.828,167.347,49.297,159.086
C01561=1023.092,47.157,-102.845,167.350,49.292,159.085
C01562=1023.098,47.406,-102.861,167.352,49.288,159.085
C01563=1023.104,47.655,-102.877,167.355,49.283,159.085
C01564=1023.110,47.905,-102.894,167.358,49.279,159.084
C01565=1023.116,48.154,-102.910,167.361,49.274,159.084
C01566=1023.122,48.403,-102.926,167.363,49.270,159.083
C01567=1023.128,48.653,-102.943,167.366,49.266,159.083
C01568=1023.133,48.903,-102.959,167.368,49.261,159.082
C01569=1023.139,49.152,-102.976,167.371,49.257,159.082
C01570=1023.145,49.401,-102.992,167.373,49.252,159.082
C01571=1023.151,49.651,-103.008,167.376,49.248,159.081
C01572=1023.157,49.900,-103.024,167.378,49.244,159.081
C01573=1023.163,50.149,-103.041,167.381,49.239,159.080
C01574=1023.169,50.399,-103.057,167.384,49.235,159.080
C01575=1023.174,50.648,-103.074,167.386,49.231,159.079
C01576=1023.180,50.898,-103.090,167.388,49.226,159.079
C01577=1023.186,51.147,-103.106,167.391,49.222,159.078
C01578=1023.192,51.396,-103.123,167.393,49.217,159.078
C01579=1023.198,51.646,-103.139,167.397,49.212,159.077
C01580=1023.204,51.895,-103.155,167.400,49.208,159.077
C01581=1023.210,52.145,-103.172,167.402,49.204,159.077
C01582=1023.215,52.395,-103.189,167.404,49.199,159.076
C01583=1023.222,52.643,-103.205,167.407,49.195,159.076
C01584=1023.228,52.893,-103.222,167.409,49.190,159.075
C01585=1023.234,53.142,-103.238,167.412,49.186,159.075
C01586=1023.240,53.391,-103.254,167.415,49.182,159.074
C01587=1023.246,53.641,-103.271,167.417,49.177,159.074
C01588=1023.251,53.890,-103.287,167.419,49.173,159.073
C01589=1023.257,54.140,-103.304,167.422,49.169,159.073
C01590=1023.263,54.389,-103.320,167.425,49.164,159.073
C01591=1023.269,54.639,-103.336,167.428,49.159,159.072
C01592=1023.275,54.887,-103.353,167.430,49.154,159.072
C01593=1023.281,55.137,-103.369,167.433,49.150,159.071
C01594=1023.287,55.387,-103.386,167.435,49.146,159.071
C01595=1023.293,55.636,-103.403,167.438,49.141,159.070
C01596=1023.299,55.886,-103.419,167.440,49.137,159.070
C01597=1023.304,56.135,-103.435,167.443,49.132,159.069
C01598=1023.310,56.384,-103.452,167.445,49.128,159.069
C01599=1023.317,56.633,-103.469,167.449,49.123,159.068
C01600=1023.323,56.882,-103.485,167.451,49.119,159.068
C01601=1023.328,57.132,-103.502,167.454,49.114,159.067
C01602=1023.334,57.382,-103.518,167.456,49.110,159.067
C01603=1023.340,57.632,-103.535,167.459,49.105,159.066
C01604=1023.347,57.880,-103.552,167.461,49.101,159.066
C01605=1023.353,58.130,-103.568,167.464,49.096,159.066
C01606=1023.359,58.379,-103.584,167.466,49.092,159.065
C01607=1023.364,58.629,-103.601,167.469,49.087,159.065
C01608=1023.371,58.878,-103.618,167.472,49.082,159.064
C01609=1023.377,59.162,-103.637,167.474,49.078,159.064
C01610=1023.384,59.446,-103.655,167.478,49.073,159.063
C01611=1023.391,59.731,-103.674,167.481,49.067,159.062
C01612=1023.398,60.015,-103.694,167.484,49.062,159.062
C01613=1023.403,60.264,-103.710,167.487,49.057,159.062
C01614=1023.409,60.514,-103.726,167.489,49.053,159.061
C01615=1023.416,60.763,-103.744,167.491,49.048,159.060
C01616=1023.422,61.012,-103.760,167.494,49.043,159.060
C01617=1023.428,61.262,-103.776,167.496,49.040,159.060
C01618=1023.433,61.511,-103.793,167.499,49.035,159.059
C01619=1023.440,61.760,-103.810,167.502,49.030,159.059
C01620=1023.446,62.010,-103.827,167.505,49.025,159.058
C01621=1023.452,62.259,-103.843,167.507,49.021,159.058
C01622=1023.458,62.508,-103.860,167.509,49.016,159.057
C01623=1023.464,62.758,-103.877,167.512,49.011,159.057
C01624=1023.470,63.008,-103.893,167.515,49.007,159.056
C01625=1023.476,63.257,-103.910,167.517,49.003,159.056
C01626=1023.482,63.506,-103.927,167.520,48.998,159.055
C01627=1023.488,63.755,-103.944,167.523,48.993,159.055
C01628=1023.494,64.005,-103.961,167.526,48.989,159.054
C01629=1023.500,64.254,-103.978,167.528,48.985,159.054
C01630=1023.505,64.504,-103.995,167.530,48.980,159.053
C01631=1023.511,64.753,-104.012,167.533,48.976,159.053
C01632=1023.517,65.003,-104.029,167.535,48.972,159.052
C01633=1023.524,65.252,-104.046,167.538,48.967,159.052
C01634=1023.529,65.501,-104.063,167.541,48.963,159.052
C01635=1023.535,65.750,-104.080,167.543,48.958,159.051
C01636=1023.542,66.000,-104.097,167.545,48.954,159.051
C01637=1023.547,66.249,-104.114,167.548,48.949,159.050
C01638=1023.552,66.499,-104.131,167.551,48.945,159.050
C01639=1023.559,66.747,-104.148,167.554,48.940,159.049
C01640=1023.564,66.998,-104.165,167.556,48.936,159.049
C01641=1023.571,67.247,-104.182,167.559,48.932,159.048
C01642=1023.576,67.496,-104.200,167.562,48.927,159.048
C01643=1023.582,67.745,-104.216,167.564,48.922,159.047
C01644=1023.588,67.995,-104.234,167.567,48.918,159.047
C01645=1023.594,68.244,-104.250,167.569,48.914,159.046
C01646=1023.600,68.493,-104.268,167.572,48.909,159.046
C01647=1023.607,68.743,-104.285,167.574,48.905,159.045
C01648=1023.612,68.992,-104.302,167.577,48.901,159.045
C01649=1023.617,69.241,-104.320,167.579,48.896,159.045
C01650=1023.624,69.491,-104.337,167.581,48.891,159.044
C01651=1023.629,69.740,-104.354,167.584,48.888,159.044
C01652=1023.635,69.989,-104.371,167.587,48.883,159.043
C01653=1023.640,70.238,-104.389,167.590,48.878,159.043
C01654=1023.647,70.488,-104.406,167.593,48.874,159.042
C01655=1023.652,70.737,-104.423,167.595,48.869,159.042
C01656=1023.658,70.987,-104.441,167.598,48.865,159.041
C01657=1023.665,71.236,-104.458,167.600,48.861,159.041
C01658=1023.670,71.486,-104.475,167.603,48.856,159.040
C01659=1023.676,71.735,-104.493,167.605,48.852,159.040
C01660=1023.682,71.984,-104.510,167.608,48.848,159.040
C01661=1023.688,72.233,-104.527,167.610,48.843,159.039
C01662=1023.693,72.483,-104.544,167.613,48.839,159.038
C01663=1023.699,72.733,-104.562,167.616,48.835,159.038
C01664=1023.705,72.981,-104.579,167.618,48.830,159.038
C01665=1023.711,73.230,-104.597,167.620,48.825,159.037
C01666=1023.717,73.480,-104.615,167.623,48.821,159.037
C01667=1023.723,73.729,-104.631,167.627,48.817,159.036
C01668=1023.729,73.978,-104.649,167.629,48.812,159.036
C01669=1023.735,74.228,-104.666,167.631,48.807,159.035
C01670=1023.740,74.477,-104.684,167.634,48.803,159.035
C01671=1023.747,74.727,-104.701,167.637,48.799,159.034
C01672=1023.753,74.976,-104.719,167.639,48.794,159.034
C01673=1023.759,75.260,-104.739,167.642,48.789,159.033
C01674=1023.766,75.544,-104.759,167.645,48.784,159.033
C01675=1023.772,75.828,-104.778,167.648,48.779,159.032
C01676=1023.780,76.112,-104.798,167.651,48.774,159.032
C01677=1023.785,76.361,-104.816,167.654,48.770,159.031
C01678=1023.791,76.611,-104.834,167.656,48.765,159.031
C01679=1023.797,76.860,-104.851,167.659,48.761,159.030
C01680=1023.803,77.110,-104.868,167.661,48.757,159.030
C01681=1023.809,77.359,-104.885,167.664,48.752,159.029
C01682=1023.814,77.608,-104.903,167.667,48.748,159.029
C01683=1023.820,77.858,-104.921,167.669,48.743,159.028
C01684=1023.826,78.107,-104.939,167.671,48.739,159.028
C01685=1023.832,78.356,-104.956,167.674,48.735,159.028
C01686=1023.838,78.605,-104.974,167.677,48.730,159.027
C01687=1023.844,78.855,-104.993,167.679,48.726,159.027
C01688=1023.850,79.104,-105.010,167.682,48.722,159.026
C01689=1023.855,79.353,-105.028,167.684,48.717,159.026
C01690=1023.861,79.602,-105.046,167.687,48.713,159.025
C01691=1023.867,79.851,-105.063,167.689,48.709,159.025
C01692=1023.873,80.101,-105.081,167.692,48.704,159.024
C01693=1023.878,80.350,-105.099,167.695,48.700,159.024
C01694=1023.884,80.600,-105.117,167.698,48.695,159.023
C01695=1023.890,80.849,-105.134,167.700,48.691,159.023
C01696=1023.896,81.098,-105.152,167.703,48.687,159.023
C01697=1023.902,81.348,-105.170,167.706,48.682,159.022
C01698=1023.907,81.597,-105.187,167.708,48.678,159.021
C01699=1023.914,81.846,-105.206,167.711,48.674,159.021
C01700=1023.919,82.095,-105.224,167.713,48.669,159.021
C01701=1023.925,82.345,-105.242,167.716,48.665,159.020
C01702=1023.931,82.594,-105.259,167.718,48.661,159.020
C01703=1023.937,82.844,-105.277,167.721,48.656,159.019
C01704=1023.942,83.093,-105.295,167.723,48.651,159.019
C01705=1023.948,83.343,-105.313,167.726,48.648,159.018
C01706=1023.954,83.591,-105.331,167.729,48.643,159.018
C01707=1023.960,83.841,-105.349,167.731,48.638,159.017
C01708=1023.965,84.090,-105.367,167.734,48.634,159.017
C01709=1023.971,84.340,-105.385,167.737,48.630,159.016
C01710=1023.977,84.589,-105.402,167.740,48.625,159.016
C01711=1023.983,84.838,-105.421,167.742,48.620,159.015
C01712=1023.989,85.087,-105.439,167.745,48.617,159.015
C01713=1023.995,85.337,-105.457,167.747,48.612,159.015
C01714=1024.000,85.586,-105.474,167.750,48.607,159.014
C01715=1024.007,85.835,-105.492,167.752,48.603,159.013
C01716=1024.012,86.084,-105.510,167.755,48.599,159.013
C01717=1024.019,86.333,-105.528,167.757,48.594,159.013
C01718=1024.024,86.583,-105.546,167.760,48.590,159.012
C01719=1024.030,86.832,-105.564,167.764,48.586,159.012
C01720=1024.037,87.081,-105.582,167.766,48.581,159.011
C01721=1024.042,87.330,-105.600,167.768,48.576,159.011
C01722=1024.048,87.580,-105.618,167.771,48.572,159.010
C01723=1024.054,87.829,-105.635,167.773,48.567,159.010
C01724=1024.060,88.078,-105.654,167.776,48.563,159.009
C01725=1024.066,88.327,-105.672,167.779,48.559,159.009
C01726=1024.072,88.577,-105.690,167.781,48.554,159.008
C01727=1024.078,88.826,-105.708,167.783,48.550,159.008
C01728=1024.084,89.075,-105.726,167.787,48.545,159.007
C01729=1024.090,89.325,-105.744,167.790,48.541,159.007
C01730=1024.095,89.574,-105.763,167.792,48.536,159.006
C01731=1024.101,89.823,-105.781,167.795,48.532,159.006
C01732=1024.107,90.073,-105.799,167.797,48.528,159.005
C01733=1024.112,90.322,-105.817,167.800,48.523,159.005
C01734=1024.118,90.572,-105.835,167.803,48.519,159.005
C01735=1024.124,90.820,-105.854,167.805,48.515,159.004
C01736=1024.130,91.070,-105.872,167.808,48.511,159.004
C01737=1024.137,91.354,-105.893,167.811,48.505,159.003
C01738=1024.144,91.638,-105.914,167.813,48.501,159.003
C01739=1024.150,91.922,-105.934,167.817,48.496,159.002
C01740=1024.156,92.206,-105.956,167.820,48.490,159.001
C01741=1024.162,92.455,-105.974,167.823,48.486,159.001
C01742=1024.168,92.704,-105.992,167.825,48.482,159.001
C01743=1024.174,92.954,-106.011,167.828,48.477,159.000
C01744=1024.180,93.204,-106.029,167.830,48.473,159.000
C01745=1024.185,93.452,-106.047,167.833,48.469,158.999
C01746=1024.191,93.702,-106.066,167.835,48.464,158.999
C01747=1024.197,93.950,-106.084,167.838,48.460,158.998
C01748=1024.203,94.200,-106.103,167.840,48.456,158.998
C01749=1024.208,94.450,-106.121,167.843,48.451,158.997
C01750=1024.214,94.698,-106.140,167.846,48.447,158.997
C01751=1024.220,94.948,-106.158,167.848,48.443,158.996
C01752=1024.226,95.197,-106.177,167.852,48.438,158.996
C01753=1024.232,95.446,-106.194,167.854,48.434,158.996
C01754=1024.238,95.695,-106.213,167.857,48.430,158.995
C01755=1024.244,95.945,-106.232,167.859,48.425,158.994
C01756=1024.249,96.194,-106.250,167.862,48.421,158.994
C01757=1024.256,96.443,-106.268,167.865,48.417,158.994
C01758=1024.261,96.693,-106.287,167.867,48.412,158.993
C01759=1024.267,96.941,-106.305,167.869,48.407,158.992
C01760=1024.273,97.191,-106.324,167.872,48.404,158.992
C01761=1024.279,97.441,-106.342,167.875,48.399,158.992
C01762=1024.285,97.690,-106.361,167.878,48.394,158.991
C01763=1024.290,97.938,-106.380,167.881,48.390,158.991
C01764=1024.296,98.188,-106.398,167.883,48.386,158.990
C01765=1024.303,98.437,-106.417,167.886,48.381,158.990
C01766=1024.308,98.686,-106.435,167.888,48.377,158.989
C01767=1024.314,98.936,-106.453,167.891,48.373,158.989
C01768=1024.320,99.185,-106.472,167.894,48.368,158.988
C01769=1024.326,99.434,-106.491,167.897,48.363,158.988
C01770=1024.332,99.683,-106.509,167.900,48.360,158.987
C01771=1024.337,99.933,-106.528,167.902,48.355,158.987
C01772=1024.343,100.182,-106.547,167.905,48.350,158.986
C01773=1024.349,100.431,-106.566,167.908,48.347,158.986
C01774=1024.354,100.680,-106.585,167.910,48.342,158.986
C01775=1024.361,100.930,-106.603,167.913,48.338,158.985
C01776=1024.366,101.179,-106.622,167.915,48.334,158.985
C01777=1024.371,101.428,-106.641,167.918,48.329,158.984
C01778=1024.378,101.677,-106.660,167.921,48.325,158.984
C01779=1024.383,101.927,-106.679,167.923,48.321,158.983
C01780=1024.389,102.176,-106.698,167.926,48.317,158.983
C01781=1024.395,102.424,-106.716,167.928,48.312,158.982
C01782=1024.400,102.675,-106.735,167.931,48.308,158.982
C01783=1024.406,102.924,-106.754,167.934,48.304,158.981
C01784=1024.412,103.173,-106.773,167.937,48.299,158.981
C01785=1024.418,103.422,-106.792,167.939,48.294,158.980
C01786=1024.423,103.671,-106.811,167.942,48.291,158.980
C01787=1024.430,103.920,-106.830,167.945,48.286,158.980
C01788=1024.435,104.170,-106.849,167.947,48.282,158.979
C01789=1024.442,104.419,-106.867,167.950,48.278,158.979
C01790=1024.447,104.668,-106.886,167.952,48.273,158.978
C01791=1024.453,104.917,-106.906,167.955,48.269,158.978
C01792=1024.459,105.166,-106.924,167.958,48.265,158.977
C01793=1024.465,105.416,-106.943,167.961,48.260,158.977
C01794=1024.470,105.664,-106.962,167.964,48.256,158.976
C01795=1024.476,105.913,-106.981,167.966,48.251,158.976
C01796=1024.482,106.164,-106.999,167.969,48.247,158.975
C01797=1024.487,106.413,-107.019,167.972,48.243,158.975
C01798=1024.494,106.662,-107.037,167.974,48.239,158.974
C01799=1024.499,106.912,-107.057,167.977,48.234,158.974
C01800=1024.504,107.160,-107.075,167.979,48.230,158.973
C01801=1024.512,107.444,-107.098,167.983,48.225,158.973
C01802=1024.519,107.729,-107.119,167.986,48.220,158.972
C01803=1024.525,108.013,-107.141,167.990,48.215,158.972
C01804=1024.532,108.296,-107.163,167.992,48.210,158.971
C01805=1024.538,108.546,-107.182,167.996,48.206,158.971
